FOR i := 1 TO fbSlotList.P_nCount BY 1 DO
	pSlot := fbSlotList.M_GetNext();
	IF pSlot > 0 THEN
		nCurrentPropIndex := nCurrentPropIndex + 1;
		refCmdData.n32Data[nCurrentPropIndex] := pSlot^.P_nNr;
		nCurrentPropIndex := nCurrentPropIndex + 1;
		refCmdData.n32Data[nCurrentPropIndex] := REAL_TO_DINT(pSlot^.P_rRelPosX);
		nCurrentPropIndex := nCurrentPropIndex + 1;
		refCmdData.n32Data[nCurrentPropIndex] := REAL_TO_DINT(pSlot^.P_rRelPosY);
		nCurrentPropIndex := nCurrentPropIndex + 1;
		refCmdData.n32Data[nCurrentPropIndex] := REAL_TO_DINT(pSlot^.P_rRelPosZ);
		nCurrentPropIndex := nCurrentPropIndex + 1;
		refCmdData.n32Data[nCurrentPropIndex] := REAL_TO_DINT(pSlot^.P_rDimWidth);
		nCurrentPropIndex := nCurrentPropIndex + 1;
		refCmdData.n32Data[nCurrentPropIndex] := REAL_TO_DINT(pSlot^.P_rDimDepth);
	END_IF		
END_FOR

nCurrentPropIndex := nCurrentPropIndex + 1;
refCmdData.n32Data[nCurrentPropIndex] := nValveNrSlot1;
nCurrentPropIndex := nCurrentPropIndex + 1;
refCmdData.n32Data[nCurrentPropIndex] := nValveNrSlot2;
nCurrentPropIndex := nCurrentPropIndex + 1;
refCmdData.n32Data[nCurrentPropIndex] := nPumpNrWaste;
nCurrentPropIndex := nCurrentPropIndex + 1;
refCmdData.n32Data[nCurrentPropIndex] := nBottleNrWaste;
END_METHOD

METHOD M_GetProcData : DINT
VAR_INPUT
	eProcDataType : E_ProcDataType;
END_VAR
END_METHOD

METHOD M_GetRectIsInnerSlot : BOOL
VAR_INPUT
	stRectArea : FB_Rectangle;
END_VAR

VAR
	pSlot : POINTER TO FB_DimSlot;
	stPoint: ST_3DPoint;
	fbRect : FB_Rectangle;
	
	
	END_VAR
//Alle Slots durchlaufen
fbSlotList.M_SetCurrentToHead();
REPEAT
	pSlot := fbSlotList.M_GetNext();
	IF pSlot > 0 THEN
		stPoint := pSlot^.P_stAbsPos;
		fbRect.X1 := stPoint.X;
		fbRect.Y1 := stPoint.Y;
		fbRect.X2 := fbRect.X1 + pSlot^.P_rDimWidth;
		fbRect.Y2 := fbRect.Y1 + pSlot^.P_rDimDepth;  
		IF F_RectInnerRect(stRectArea,fbRect) THEN
			M_GetRectIsInnerSlot := TRUE;
			RETURN;
		END_IF
	END_IF
UNTIL pSlot = 0
END_REPEAT
END_METHOD

METHOD M_GetSlot : POINTER TO FB_Slot
VAR_INPUT
	nSlotNr : UINT;
END_VAR
M_GetSlot := fbSlotList.M_GetAtNr(nSlotNr);
END_METHOD

METHOD M_GetSlotFromChild : POINTER TO FB_Slot
VAR_INPUT
	pObject : POINTER TO FB_Object;
END_VAR

VAR
	pSlot : POINTER TO FB_Slot;
END_VAR
//Die SlotList iterieren und vergleichen ob Objekte übereinstimmen
fbSlotList.M_SetCurrentToHead();
REPEAT
	pSlot := fbSlotList.M_GetNext();
	IF pSlot > 0 THEN
		IF pSlot^.P_pChild = pObject THEN
			M_GetSlotFromChild := pSlot;
			EXIT;
		END_IF
	END_IF
UNTIL pSlot = 0
END_REPEAT
END_METHOD

METHOD M_Reset
bError := FALSE;
bBusy := FALSE;
eCurrentState := E_MachineState.MACHINESTATE_Idle;
END_METHOD

METHOD M_SetAllProps : ERRORID
VAR_INPUT
	refCmdData : REFERENCE TO  ST_CmdData;
END_VAR

VAR
	i : UINT;
END_VAR
M_SetAllProps := SUPER^.M_SetAllProps(refCmdData);

IF M_SetAllProps > 0 THEN
	RETURN;
END_IF

//Slots parametrieren
nCurrentPropIndex := nCurrentPropIndex + 1;
nFirstSlotPropIndex := nCurrentPropIndex;
nNumberOfSlots := DINT_TO_UINT(refCmdData.n32Data[nCurrentPropIndex]);

//Falls SlotList noch nicht existiert, dann neue erstellen
IF fbSlotList.P_nCount = 0 THEN
	FOR i:= 1 TO nNumberOfSlots BY 1 DO
		pSlot := __NEW(FB_DimSlot(pOwner := THIS));
		fbSlotList.M_Add(pSlot);
		nCurrentPropIndex := nCurrentPropIndex + 1;
		pSlot^.P_nNr := DINT_TO_USINT(refCmdData.n32Data[nCurrentPropIndex]);
		nCurrentPropIndex := nCurrentPropIndex + 1;
		pSlot^.P_rRelPosX := DINT_TO_REAL(refCmdData.n32Data[nCurrentPropIndex]);
		nCurrentPropIndex := nCurrentPropIndex + 1;
		pSlot^.P_rRelPosY := DINT_TO_REAL(refCmdData.n32Data[nCurrentPropIndex]);
		nCurrentPropIndex := nCurrentPropIndex + 1;
		pSlot^.P_rRelPosZ := DINT_TO_REAL(refCmdData.n32Data[nCurrentPropIndex]);
		nCurrentPropIndex := nCurrentPropIndex + 1;
		pSlot^.P_rDimWidth := DINT_TO_REAL(refCmdData.n32Data[nCurrentPropIndex]);
		nCurrentPropIndex := nCurrentPropIndex + 1;
		pSlot^.P_rDimDepth := DINT_TO_REAL(refCmdData.n32Data[nCurrentPropIndex]);
	END_FOR
ELSE
	IF nNumberOfSlots <> fbSlotList.P_nCount THEN	//Anzahl der Slots dürfen sich nicht ändern
		M_SetAllProps := E_ErrorIdObjMgmt.ERRORID_ChangeNoOfSlotsNotAllowed;
		RETURN;		
	END_IF

	FOR i:= 1 TO nNumberOfSlots BY 1 DO
		nCurrentPropIndex := nCurrentPropIndex + 1;
		pSlot := fbSlotList.M_GetAtNr(DINT_TO_USINT(refCmdData.n32Data[nCurrentPropIndex]));
		IF pSlot > 0 THEN
			nCurrentPropIndex := nCurrentPropIndex + 1;
			pSlot^.P_rRelPosX := DINT_TO_REAL(refCmdData.n32Data[nCurrentPropIndex]);
			nCurrentPropIndex := nCurrentPropIndex + 1;
			pSlot^.P_rRelPosY := DINT_TO_REAL(refCmdData.n32Data[nCurrentPropIndex]);
			nCurrentPropIndex := nCurrentPropIndex + 1;
			pSlot^.P_rRelPosZ := DINT_TO_REAL(refCmdData.n32Data[nCurrentPropIndex]);
			nCurrentPropIndex := nCurrentPropIndex + 1;
			pSlot^.P_rDimWidth := DINT_TO_REAL(refCmdData.n32Data[nCurrentPropIndex]);
			nCurrentPropIndex := nCurrentPropIndex + 1;
			pSlot^.P_rDimDepth := DINT_TO_REAL(refCmdData.n32Data[nCurrentPropIndex]);
		ELSE
			M_SetAllProps := 222;
			RETURN;
		END_IF	
	END_FOR
END_IF
nLastSlotPropIndex := nCurrentPropIndex;
nNoOfProps := nCurrentPropIndex + 1;

nCurrentPropIndex := nCurrentPropIndex + 1;
nSpecPropIndex := nCurrentPropIndex;

nValveNrSlot1 := DINT_TO_USINT(refCmdData.n32Data[nCurrentPropIndex]);
IF NOT (nValveNrSlot1 > 0 AND nValveNrSlot1 <= cNoOfValves) THEN
	M_SetAllProps := E_ErrorIdObjMgmt.ERRORID_InvalidValveNumber;
	RETURN;
END_IF

nCurrentPropIndex := nCurrentPropIndex + 1;
nValveNrSlot2 := DINT_TO_USINT(refCmdData.n32Data[nCurrentPropIndex]);
IF NOT (nValveNrSlot1 > 0 AND nValveNrSlot1 <= cNoOfValves) THEN
	M_SetAllProps := E_ErrorIdObjMgmt.ERRORID_InvalidValveNumber;
	RETURN;
END_IF

nCurrentPropIndex := nCurrentPropIndex + 1;
nPumpNrWaste := DINT_TO_USINT(refCmdData.n32Data[nCurrentPropIndex]);
IF NOT (nPumpNrWaste > 0 AND nPumpNrWaste <= cNoOfPumps) THEN
	M_SetAllProps := E_ErrorIdObjMgmt.ERRORID_InvalidPumpNumber;
	RETURN;
END_IF

nCurrentPropIndex := nCurrentPropIndex + 1;
nBottleNrWaste := DINT_TO_USINT(refCmdData.n32Data[nCurrentPropIndex]);
IF NOT (nBottleNrWaste > 0 AND nBottleNrWaste <= cNoOfWasteBottles) THEN
	M_SetAllProps := E_ErrorIdObjMgmt.ERRORID_InvalidWastebottle;
	RETURN;
END_IF

nNoOfProps := nCurrentPropIndex + 1;
END_METHOD

METHOD M_SetSingleProp : ERRORID
VAR_INPUT
	refCmdData : REFERENCE TO  ST_CmdData;
END_VAR

VAR
	i : UINT;
	nIndex					: UINT;
	nIndexRinseChannels	 	: UINT;
	nIndexWashPoints 	 	: UINT;
	nIndexRestProps 	 	: UINT;
END_VAR
(*nIndexRinseChannels := nSpecPropIndex;
nIndexWashPoints := nIndexRinseChannels + nNoOfRinseChannels * 5 + 1;
nIndexRestProps := nIndexWashPoints + nNoOfWashPoints * 4 + 1;

//Section: RinseChannels
IF refCmdData.aHeader[1] > nIndexRinseChannels AND refCmdData.aHeader[1] < nIndexWashPoints THEN
	FOR i:= 1 TO nNoOfRinseChannels BY 1 DO
		//ersten Index innerhalb der Section ermitteln
		nIndex := nIndexRinseChannels + ((i - 1) * 5) + 1;
		IF refCmdData.aHeader[1] = nIndex THEN	//PumpNr
			IF refCmdData.n32Data[0] >= 0 AND refCmdData.n32Data[0] <= cNoOfPumps THEN
				aStRinseChannels[i].nPumpNr := DINT_TO_USINT(refCmdData.n32Data[0]);
			ELSE
				M_SetSingleProp := E_ErrorIdCmd.ERRORID_InvalidPumpNr;
				RETURN;
			END_IF
			RETURN;
		ELSIF refCmdData.aHeader[1] = nIndex + 1 THEN	//ValveNr
			IF refCmdData.n32Data[0] >= 0 AND refCmdData.n32Data[0] <= cNoOfValves THEN
				aStRinseChannels[i].nValveNr := DINT_TO_USINT(refCmdData.n32Data[0]);
			ELSE
				M_SetSingleProp := E_ErrorIdObjMgmt.ERRORID_InvalidValveNumber;
				RETURN;
			END_IF
		ELSIF refCmdData.aHeader[1] = nIndex + 2 THEN	//StartSpeed in %
			aStRinseChannels[i].nStartSpeed := DINT_TO_USINT(refCmdData.n32Data[0]);	
		ELSIF refCmdData.aHeader[1] = nIndex + 3 THEN	//RatedSpeed in %
			aStRinseChannels[i].nRatedSpeed := DINT_TO_USINT(refCmdData.n32Data[0]);
		ELSIF refCmdData.aHeader[1] = nIndex + 4 THEN	//StartTime in ms
			aStRinseChannels[i].nStartTime := DINT_TO_UINT(refCmdData.n32Data[0]);
		END_IF		
	END_FOR
//Section: Washpoints	
ELSIF refCmdData.aHeader[1] > nIndexWashPoints AND refCmdData.aHeader[1] < nIndexRestProps THEN
	FOR i:= 1 TO nNoOfWashPoints BY 1 DO
		//ersten Index innerhalb der Section ermitteln
		nIndex := nIndexWashPoints + ((i - 1) * 4) + 1;
		IF refCmdData.aHeader[1] = nIndex THEN
			aStWashPoints[i].X := DINT_TO_REAL(refCmdData.n32Data[0]);
		ELSIF refCmdData.aHeader[1] = nIndex + 1 THEN
			aStWashPoints[i].Y := DINT_TO_REAL(refCmdData.n32Data[0]);
		ELSIF refCmdData.aHeader[1] = nIndex + 2 THEN
			aStWashPoints[i].Z := DINT_TO_REAL(refCmdData.n32Data[0]);
		ELSIF refCmdData.aHeader[1] = nIndex + 3 THEN
			M_SetSingleProp := E_ErrorIdCmd.ERRORID_InvalidProperty;
		END_IF			
	END_FOR
//Restliche Props
ELSIF refCmdData.aHeader[1] >= nIndexRestProps AND refCmdData.aHeader[1] < nNoOfProps THEN
	CASE (refCmdData.aHeader[1] - nIndexRestProps) OF
		0: //PumpNrWaste
			IF refCmdData.n32Data[0] > 0 AND refCmdData.n32Data[0] <= cNoOfPumps THEN
				nPumpNrWastePump := DINT_TO_USINT(refCmdData.n32Data[0]);
			ELSE
				M_SetSingleProp := E_ErrorIdCmd.ERRORID_InvalidPumpNr;
			END_IF			
		1: //LiquidBottle
			IF refCmdData.n32Data[0] > 0 AND refCmdData.n32Data[0] <= cNoOfLiquidBottles THEN
				nSysLiquidBottle := DINT_TO_USINT(refCmdData.n32Data[0]);
			ELSE
				M_SetSingleProp := E_ErrorIdObjMgmt.ERRORID_InvalidLiquidbottle;
			END_IF			
		2: //WasteBottle
			IF refCmdData.n32Data[0] > 0 AND refCmdData.n32Data[0] <= cNoOfWasteBottles THEN
				nWasteBottle := DINT_TO_USINT(refCmdData.n32Data[0]);
			ELSE
				M_SetSingleProp := E_ErrorIdObjMgmt.ERRORID_InvalidWastebottle;
			END_IF
		3: //ValveNrDrying (Trockendusche für pH Elektrode)
			IF refCmdData.n32Data[0] >= 0 AND refCmdData.n32Data[0] <= cNoOfValves THEN
				nValveNrAirShower := DINT_TO_USINT(refCmdData.n32Data[0]);
			ELSE
				M_SetSingleProp := E_ErrorIdObjMgmt.ERRORID_InvalidValveNumber;
			END_IF			
	END_CASE	
ELSE
	M_SetSingleProp := SUPER^.M_SetSingleProp(refCmdData);
END_IF*)
END_METHOD

METHOD M_Stop : ERRORID
VAR_INPUT
END_VAR
IF bSuckOff AND nStateA_SuckOff < 70 THEN
	nStateA_SuckOff:= 70;
END_IF
END_METHOD

END_FUNCTION_BLOCK

// ---- Objects/Targets/Active/FB_ActiveTarget.TcPOU
FUNCTION_BLOCK FB_ActiveTarget EXTENDS FB_TargetBase IMPLEMENTS I_Device
VAR_INPUT
END_VAR
VAR_OUTPUT
END_VAR
VAR
	bInitFB			: BOOL := TRUE;
	nNotifyId		: UINT;
	bError			: BOOL;
	nErrorId		: ERRORID;
	bCanceled		: BOOL;
	bStop			: BOOL;
	bBusy			: BOOL;
	eCurrentState	: E_MachineState := E_MachineState.MACHINESTATE_Idle;
	stError			: ST_Error;
	bIsInit			: BOOL;	
	stProcessData	: ST_ObjectProcData;
	eCurrentAction	: E_Action;
	
	//Verkettete Liste für BasicActions
	fbList				: FB_LinkedListCtrl;
	hList				: T_HLINKEDLIST;
	aNodes           	: ARRAY[0..4] OF T_LinkedListEntry;
	getValue			: PVOID;
	getPosPtr       	: POINTER TO T_LinkedListEntry := 0;
	
	
	//Action: "Init"
	bInit				: BOOL;				//Action A_Init() aktiv setzen
	nStateA_Init		: USINT;			//State von A_Init()
	bFlagA_Init			: BOOL := TRUE;		//Hilfsflag A_Init()
	
	//Action: Stop
	nStateA_Stop		: USINT;	//Statemachine von A_Stop()
	bStopAllOnError		: BOOL;
	
	//Action: "Reset"
	nStateA_Reset		: USINT;	//Statemachine von A_Reset();	
END_VAR

METHOD M_CancelAction
VAR_INPUT
	eAction	: E_Action;
END_VAR
END_METHOD

METHOD M_CheckProcDataType : BOOL
VAR_INPUT
	eProcDataType : E_ProcDataType;
END_VAR
END_METHOD

METHOD M_ExeAction : ERRORID
VAR_INPUT
	refActionData	: REFERENCE TO ST_ActionData;
END_VAR
END_METHOD

METHOD M_GetActionBusy : BOOL
VAR_INPUT
	eAction	: E_Action;
END_VAR
END_METHOD

METHOD M_GetAllProps : ERRORID
VAR_INPUT
	refCmdData : REFERENCE TO ST_CmdData;
END_VAR
M_GetAllProps := SUPER^.M_GetAllProps(refCmdData);
refCmdData.aHeader[2] := nNotifyId;
END_METHOD

METHOD M_GetDevice : I_Device
VAR_INPUT
END_VAR
M_GetDevice := THIS^;
END_METHOD

METHOD M_GetProcData : DINT
VAR_INPUT
	eProcDataType : E_ProcDataType;
END_VAR
END_METHOD

METHOD M_Reset
bBusy := TRUE;
eCurrentState := E_MachineState.MACHINESTATE_Reset;
END_METHOD

METHOD M_Stop : ERRORID
//Stop braucht nur ausgeführt werden, wenn irgendwas aktiv ist
IF NOT bStop AND eCurrentState = E_MachineState.MACHINESTATE_Active THEN
	bStop := TRUE;
	fbList.A_AddHeadValue(hList := hList, putValue := E_Action.ACTION_Stop);
END_IF
END_METHOD

PROPERTY P_bBusy : BOOL
GET
P_bBusy := bBusy;
END_GET
END_PROPERTY

PROPERTY P_bCanceled : BOOL
GET
P_bCanceled := bCanceled;
END_GET
END_PROPERTY

PROPERTY P_bError : BOOL
GET
P_bError := bError;
END_GET
END_PROPERTY

PROPERTY P_bIsInit : BOOL
GET
P_bIsInit := bIsInit;
END_GET
END_PROPERTY

PROPERTY P_bStopAllOnError : BOOL
GET
P_bStopAllOnError := bStopAllOnError;
END_GET
END_PROPERTY

PROPERTY P_eCurrentState : E_MachineState
GET
P_eCurrentState := eCurrentState;
END_GET
END_PROPERTY

PROPERTY P_nErrorId : ERRORID
GET
P_nErrorID := nErrorID;
END_GET
END_PROPERTY

PROPERTY P_nNotifyId : UINT
GET
P_nNotifyId := nNotifyId;
END_GET
SET
nNotifyId := P_nNotifyId;
END_SET
END_PROPERTY

PROPERTY P_pObject : POINTER TO FB_Object
GET
P_pObject := THIS;
END_GET
END_PROPERTY

PROPERTY P_stError : ST_Error
GET
P_stError := stError;
END_GET
END_PROPERTY

END_FUNCTION_BLOCK

// ---- Objects/FB_DimSlot.TcPOU
{attribute 'enable_dynamic_creation'}
FUNCTION_BLOCK FB_DimSlot EXTENDS FB_Slot
VAR_INPUT
END_VAR
VAR_OUTPUT
END_VAR
VAR
	stDimension : ST_3DDimension;
END_VAR

PROPERTY P_rDimDepth : REAL
GET
P_rDimDepth := stDimension.Depth;
END_GET
SET
stDimension.Depth := P_rDimDepth;
END_SET
END_PROPERTY

PROPERTY P_rDimHeight : REAL
GET
P_rDimHeight := stDimension.Height;
END_GET
SET
stDimension.Height := P_rDimHeight;
END_SET
END_PROPERTY

PROPERTY P_rDimWidth : REAL
GET
P_rDimWidth := stDimension.Width;
END_GET
SET
stDimension.Width := P_rDimWidth;
END_SET
END_PROPERTY

PROPERTY P_stDimension : ST_3DDimension
GET
P_stDimension := stDimension;
END_GET
SET
stDimension := P_stDimension;
END_SET
END_PROPERTY

END_FUNCTION_BLOCK

// ---- Objects/F_RectInnerRect.TcPOU
FUNCTION F_RectInnerRect : BOOL
VAR_INPUT
	stRect1 : FB_Rectangle;
	stRect2 : FB_Rectangle;
END_VAR
VAR
END_VAR

//Rechteck1 innerhalb Rechteck2?
F_RectInnerRect :=

(stRect1.X1 >= stRect2.X1) AND 
(stRect1.X1 <= stRect2.X2) AND
(stRect1.X2 >= stRect2.X1) AND
(stRect1.X2 <= stRect2.X2) AND

(stRect1.Y1 >= stRect2.Y1) AND 
(stRect1.Y1 <= stRect2.Y2) AND
(stRect1.Y2 >= stRect2.Y1) AND
(stRect1.Y2 <= stRect2.Y2);

END_FUNCTION

// ---- Functions/F_SynchronizeSpeeds.TcPOU
FUNCTION F_SynchronizeSpeeds : ARRAY[0..1] OF REAL;
VAR_INPUT
	rSpeedSum 	: REAL;
	rDistance1 	: REAL;
	rDistance2 	: REAL;
END_VAR
VAR_IN_OUT
	rSpeed1 : REAL;
	rSpeed2 : REAL;
END_VAR
VAR
	rDistSum : REAL;
	rTime : REAL;
END_VAR

//Gesamtweg (Vektor) berechnen
rDistSum := SQRT(rDistance1 * rDistance1 + rDistance2 * rDistance2);
rTime := rDistSum / rSpeedSum;
rSpeed1 := ABS(rDistance1 / rTime);
rSpeed2 := ABS(rDistance2 / rTime);

END_FUNCTION

// ---- Hardware/MultiZ/FB_ZM_Jog.TcPOU
FUNCTION_BLOCK FB_ZM_Jog
VAR_INPUT
	bJogForward		: BOOL;
	bJogBackwards	: BOOL;
	bClock			: BOOL;
	bInching		: BOOL;	//Betriebsart Incremental, es wird um die relative Position bewegt
	pfbZAxisRef		: POINTER TO FB_ZAxisRef;
	rSpeed			: REAL;	//Geschwindigkeit
	rDistance		: REAL;	//relative Distanz, um die in der Betriebsart Incremental verfahren wird
END_VAR

VAR_OUTPUT
	bBusy			: BOOL;
	bError			: BOOL;
	nErrorID		: ERRORID;
END_VAR

VAR
	rTrig1			: R_TRIG;
	fTrig1			: F_TRIG;
	_bClock			: BOOL;
	timeOut			: TON;		//für Betriebsart "Standard" , wenn in dieser Zeitspanne keine neue Flanke kommt, dann Stop
								//verhindert, dass bei einer Unterbrechung der Kommunikation, die Achse unkontrolliert bis an das jeweilige Ende fährt

	bCurrDirForw		: BOOL;		
	bCurrDirBackw		: BOOL;		
	nState				: USINT;
	timeOutErr			: TON;
	rTargetPosition		: REAL;
	nStopReason			: USINT;	//1:regulär 2:timeout clock 3:Richtungswechsel
	nCountStopDirChange : USINT;
END_VAR

IF pfbZAxisRef = 0 THEN
	nErrorId := E_ErrorIdMultiZ.ERRORID_InvalidZChannel;
	bError := TRUE;
	nState := 99;	//go in errorstate		
	RETURN;	
END_IF

//Wird Achse momentan von anderem Movebaustein genutzt?
IF (pfbZAxisRef^.pCurrentFb > 0) AND (pfbZAxisRef^.pCurrentFb <> THIS) THEN //wird von anderem FB genutzt
	RETURN;
END_IF


pfbZAxisRef^.stStatus.bIsMoving := TRUE;

bBusy := TRUE;
fTrig1(CLK:= bJogForward OR bJogBackwards);	//negative Flanke von bJogForward bzw bJogBackwards stoppt
timeOut();	//in der Betriebsart "Standard" muss innerhalb einer gewissen Zeitspanne eine erneute positive Flanke am Eingang kommen, sonst "STOP"

IF pfbZAxisRef^.stInput.nStatus.3 THEN	//Error im Antrieb
	pfbZAxisRef^.stStatus.bError := TRUE;
	bBusy := FALSE;
	pfbZAxisRef^.stOutput.nMode := 0;
	pfbZAxisRef^.stOutput.nCtrl := 0;
	nErrorID := F_MultiZError_TO_ErrorId(pfbZAxisRef^.stInput.nError);
	timeOut(IN:= FALSE);
	bError := TRUE;
	bCurrDirForw := FALSE;
	bCurrDirBackw := FALSE;
	nState := 99;
END_IF

IF timeOutErr.Q THEN
	timeOutErr(IN:= FALSE);
	pfbZAxisRef^.stOutput.nMode := 0;
	pfbZAxisRef^.stOutput.nCtrl := 0;
	CASE nState OF
		2:	//Timeout wait for setpointacknowledge
			nErrorId := E_ErrorIdMultiZ.ERRORID_ToWaitSetPointAck;
		3: //Timeout wait for targetreached
			nErrorId := E_ErrorIdMultiZ.ERRORID_ToWaitTrgtReached;
		6: //Timeout wait for stop
			nErrorId := E_ErrorIdMultiZ.ERRORID_ToWaitStop;
	ELSE
		nErrorId := E_ErrorIdMultiZ.ERRORID_UnknownError;			
	END_CASE
	pfbZAxisRef^.stOutput.nMode := 0;
	pfbZAxisRef^.stOutput.nCtrl := 0;
	bCurrDirForw := FALSE;
	bCurrDirBackw := FALSE;
	bBusy := FALSE;
	bError := TRUE;
	nState := 99;	//go in errorstate
	RETURN;
END_IF

IF NOT bInching AND (bJogForward OR bJogBackwards) THEN	//Betriebsart "Continous"
	IF bClock <> _bClock THEN	//Clock, welcher innerhalb des Timeouts toggeln muss
		rTrig1(CLK:= TRUE);
		_bClock := bClock;
		timeOut(IN:= FALSE);
		timeOut(IN:= TRUE, PT:= T#550MS);		
		//wenn gerade in Move und Richtungsumkehr, dann vorher stoppen
		IF bCurrDirForw AND bJogBackwards THEN	//Richtungsumkehr, stoppen
			nStopReason := 3;
			nState := 5;
		ELSIF bCurrDirBackw AND bJogForward THEN	//Richtungsumkehr, stoppen
			nStopReason := 3;
			nState := 5;
		ELSE
			//Aktuelle Richtung setzen
			IF bJogForward THEN
				bCurrDirForw := TRUE;
				bCurrDirBackw := FALSE;
			ELSIF bJogBackwards THEN
				bCurrDirForw := FALSE;
				bCurrDirBackw := TRUE;
			END_IF			
		END_IF
	ELSE
		IF timeOut.Q THEN	//TiomeOut -> Stoppen
			timeOut(IN:= FALSE);
			nStopReason := 2;
			nstate := 5;	//Stoppen
		END_IF
	END_IF
END_IF

IF fTrig1.Q AND nState > 0  THEN
	timeOut(IN:= FALSE);
	nStopReason := 1;
	nstate := 5;	//Stoppen
END_IF

CASE nState OF
	0:	IF rTrig1.Q THEN
			timeOut(IN:= TRUE, PT:= T#500MS);	//in dieser Zeitzspanne muss eine erneute Flanke kommen, sonst "STOP"
		END_IF
		pfbZAxisRef^.pCurrentFb := THIS; 
		//Geschwindigkeit setzen
		pfbZAxisRef^.stOutput.nVelo := REAL_TO_DINT(rSpeed);
		//Betriebsart Positionsmodus setzen
		pfbZAxisRef^.stOutput.nMode := 1;
		pfbZAxisRef^.stOutput.nCtrl.2 := TRUE; //Relativ

		IF bJogForward THEN //nach oben
			rTargetPosition := pfbZAxisRef^.P_rCurrentPos + rDistance;
			IF rTargetPosition > pfbZAxisRef^.P_rMaxPos THEN
				//Distance anpassen
				rDistance := pfbZAxisRef^.P_rMaxPos - pfbZAxisRef^.P_rCurrentPos;
			END_IF
		ELSE //nach unten
			rTargetPosition := pfbZAxisRef^.P_rCurrentPos - rDistance;
			IF rTargetPosition < pfbZAxisRef^.P_rMinPos THEN
				//Distance anpassen
				rDistance := pfbZAxisRef^.P_rMinPos - pfbZAxisRef^.P_rCurrentPos;
			ELSE
				rDistance := rDistance * -1.0;
			END_IF
		END_IF

		pfbZAxisRef^.P_rRelTargetPos := rDistance;
		
		//Zielposition in Abhängigkeit von Betriebart setzen
		IF NOT bInching THEN	//Betriebsart "Standard" (Continous)
			IF bJogForward THEN //nach oben
				bCurrDirForw := TRUE;
				bCurrDirBackw := FALSE;
			ELSIF bJogBackwards THEN
				bCurrDirForw := FALSE;
				bCurrDirBackw := TRUE;
			END_IF
		END_IF
		
		//Workaround, da FB zweimal im Zyklus aufgerufen wird und Ctrl und Pos im geichen Zyklus auf den CAN-Bus geht
		nState := 10;
		
	1:	//Fahrauftrag starten
		pfbZAxisRef^.stOutput.nCtrl.0 := TRUE;
		nState := 2;
		
	10:	nState := 1;

	2:	//SetpointAcknowledge?
		//Hier könnte es zu einem TimeoutSetpointACK kommen, wenn durch FB_ZMStop Stop das StatusBit nicht kommt
		IF pfbZAxisRef^.stInput.nStatus.1 THEN
			pfbZAxisRef^.stOutput.nCtrl.0 := FALSE;	//Fahrauftrag zuücksetzen
			nState := 3;
			timeOutErr(IN:= FALSE);
		ELSE
			timeOutErr(IN:= TRUE, PT:= T#500MS);
		END_IF
		
	3:	//TargetReached?
		IF pfbZAxisRef^.stInput.nStatus.0 THEN
			rTrig1(CLK:= FALSE);
			_bClock := FALSE;
			nState := 0;	//aktuelle Postion holen
			bBusy := FALSE;
		END_IF
		
	5:	//Stoppen
		pfbZAxisRef^.stOutput.nCtrl.1 := TRUE;	//Stopbit setzen
		pfbZAxisRef^.stOutput.nCtrl.0 := FALSE;	//Fahrauftrag zurücksetzen
		timeOutErr(IN:= FALSE);
 		bCurrDirForw := FALSE;
		bCurrDirBackw := FALSE;		
		nState := 6;
		
	6:	//Stopbit gesetzt?
		IF pfbZAxisRef^.stInput.nStatus.2 THEN
			timeOutErr(IN:= FALSE);
			pfbZAxisRef^.stOutput.nCtrl.1 := FALSE;	//Stopbit zurücksetzen	
			
			pfbZAxisRef^.stOutput.nMode := 0;
				//aus welchem Grund wurde gestoppt?
			IF nStopReason = 1 THEN	//regulär gestoppt
				nState := 0;	//Aktuelle Position holen
				bBusy := FALSE;
			ELSIF nStopReason = 2 THEN //Stop durch timeout
				nState := 0;	//Aktuelle Position holen
				bBusy := FALSE;
			ELSIF nStopReason = 3 THEN //Stop durch Richtungswechsel
				_bClock := NOT _bClock;
				nCountStopDirChange := nCountStopDirChange + 1;
				nState := 0;
			END_IF
		ELSE
			timeOutErr(IN:= TRUE, PT:= T#1000MS);
		END_IF
END_CASE

IF NOT bBusy THEN
	IF pfbZAxisRef^.pCurrentFb = THIS THEN
		pfbZAxisRef^.pCurrentFb := 0;
		pfbZAxisRef^.stStatus.bIsMoving := FALSE;	
	END_IF	
END_IF

METHOD M_Reset
VAR_INPUT
END_VAR
timeOut(IN:= FALSE);
timeOutErr(IN:= FALSE);
rTrig1(CLK:= FALSE);
fTrig1(CLK:= FALSE);
_bClock := FALSE;
bError := FALSE;
nErrorID := 0;
nState := 0;
IF pfbZAxisRef^.pCurrentFb = THIS THEN
	pfbZAxisRef^.pCurrentFb := 0;
	pfbZAxisRef^.stStatus.bIsMoving := FALSE;	
END_IF
END_METHOD

END_FUNCTION_BLOCK

// ---- GCode/FB_Cuboid.TcPOU
FUNCTION_BLOCK FB_Cuboid
VAR_INPUT
END_VAR
VAR_OUTPUT
END_VAR
VAR
	stRefPoint : ST_3DPoint;
	//die  4 Eckpunkte
	aPointsBottom : ARRAY[0..3] OF ST_3DPoint;
	aPointsTop : ARRAY[0..3] OF ST_3DPoint;
	lrAngle: LREAL;	//Verdrehung um Z-Achse
END_VAR

METHOD M_IsPointInnerXY : BOOL
VAR_INPUT
	stTestPoint : ST_3DPoint;
END_VAR
VAR
	A : REAL;	//Fläche
	i : USINT;
	p1 : ST_2DPoint;
	p2 : ST_2DPoint;
	bFlag : BOOL;	
END_VAR
M_IsPointInnerXY := TRUE;
//jeweils mit allen 4 Seiten des Vierecks und dem Testpunkt ein Dreieck bilden und dessen Flächeninhalt berechen (Vektorprodukt)
FOR i := 0 TO 3 BY 1 DO
	p1.X := aPointsBottom[i].X;
	p1.Y := aPointsBottom[i].Y;
	IF i = 3 THEN
		p2.X := aPointsBottom[0].X;
		p2.Y := aPointsBottom[0].Y;
	ELSE
		p2.X := aPointsBottom[i+1].X;
		p2.Y := aPointsBottom[i+1].Y;
	END_IF
	A := 0.5 * (p1.X*p2.Y + p2.X*stTestPoint.Y + stTestPoint.X*p1.Y - p2.X*P1.Y - stTestPoint.X*p2.Y - p1.X*stTestPoint.y);
	IF A < 0.0 THEN
		M_IsPointInnerXY := FALSE;
		RETURN;
	END_IF
END_FOR
END_METHOD

METHOD M_SetDimension
VAR_INPUT
	lrX_Min : LREAL;
	lrX_Max : LREAL;
	lrY_Min : LREAL;
	lrY_Max : LREAL;
	lrZ_Min : LREAL;
	lrZ_Max : LREAL;
END_VAR
VAR
	i : USINT;
END_VAR
//in XY den Bereich etwas vergrößern (Rundungsfehler und Encoderschwankungen)
aPointsBottom[0].X := stRefPoint.X + LREAL_TO_REAL(lrX_Min) - 500.0;
aPointsBottom[0].Y := stRefPoint.Y + LREAL_TO_REAL(lrY_Min) - 500.0;
aPointsBottom[0].Z := stRefPoint.Z + LREAL_TO_REAL(lrZ_Min);

aPointsBottom[1].X := stRefPoint.X + LREAL_TO_REAL(lrX_Max) + 500.0;
aPointsBottom[1].Y := stRefPoint.Y + LREAL_TO_REAL(lrY_Min) - 500.0;
aPointsBottom[1].Z := stRefPoint.Z + LREAL_TO_REAL(lrZ_Min);

aPointsBottom[2].X := stRefPoint.X + LREAL_TO_REAL(lrX_Max) + 500.0;
aPointsBottom[2].Y := stRefPoint.Y + LREAL_TO_REAL(lrY_Max) + 500.0;
aPointsBottom[2].Z := stRefPoint.Z + LREAL_TO_REAL(lrZ_Min);

aPointsBottom[3].X := stRefPoint.X + LREAL_TO_REAL(lrX_Min) - 500.0;
aPointsBottom[3].Y := stRefPoint.Y + LREAL_TO_REAL(lrY_Max) + 500.0;
aPointsBottom[3].Z := stRefPoint.Z + LREAL_TO_REAL(lrZ_Min);

//Alle 4 Punkte drehen
FOR i := 0 TO 3 BY 1 DO
	aPointsBottom[i] := F_RotatePoint(aPointsBottom[i],stRefPoint,lrAngle);
	aPointsTop[i] := aPointsBottom[i];
 	aPointsTop[i].Z := stRefPoint.Z + LREAL_TO_REAL(lrZ_Max);
END_FOR
END_METHOD

PROPERTY P_lrAngle : LREAL
SET
lrAngle := P_lrAngle;
END_SET
END_PROPERTY

PROPERTY P_rXMax : REAL
GET
P_rXMax := MAX(MAX(MAX(aPointsBottom[0].X,aPointsBottom[1].X),aPointsBottom[2].X),aPointsBottom[3].X);
END_GET
END_PROPERTY

PROPERTY P_rXMin : REAL
GET
P_rXMin := MIN(MIN(MIN(aPointsBottom[0].X,aPointsBottom[1].X),aPointsBottom[2].X),aPointsBottom[3].X);
END_GET
END_PROPERTY

PROPERTY P_rYMax : REAL
GET
P_rYMax := MAX(MAX(MAX(aPointsBottom[0].Y,aPointsBottom[1].Y),aPointsBottom[2].Y),aPointsBottom[3].Y);
END_GET
END_PROPERTY

PROPERTY P_rYMin : REAL
GET
P_rYMin := MIN(MIN(MIN(aPointsBottom[0].Y,aPointsBottom[1].Y),aPointsBottom[2].Y),aPointsBottom[3].Y);
END_GET
END_PROPERTY

PROPERTY P_rZMax : REAL
GET
P_rZMax := aPointsTOP[0].Z;
END_GET
END_PROPERTY

PROPERTY P_rZMin : REAL
GET
P_rZMin := aPointsBottom[0].Z;
END_GET
END_PROPERTY

PROPERTY P_stRefPoint : ST_3DPoint
GET
P_stRefPoint := stRefPoint;
END_GET
SET
stRefPoint := P_stRefPoint;
END_SET
END_PROPERTY

END_FUNCTION_BLOCK

// ---- Objects/F_RotatePoint.TcPOU
FUNCTION F_RotatePoint : ST_3DPoint //Rotiert einen Punkt um einen Mittelpunkt in XY-Ebene
VAR_INPUT
	stPoint 	: ST_3DPoint;	//zu rotierender Punkt
	stPointM 	: ST_3DPoint;	//Mittelpunkt
	lrAngle 		: LREAL;	//Drehwinkel
END_VAR
VAR
	lrAngleRad 	: LREAL; //Winkel im Bogenmaß
	stLocVector : ST_2DPoint;
END_VAR

//Ortsvektor von Punkt bilden 
stLocVector.X := stPoint.X - stPointM.X;
stLocVector.Y := stPoint.Y - stPointM.Y;

lrAngleRad := DEG_TO_RAD(lrAngle);
F_RotatePoint.X := LREAL_TO_REAL(stLocVector.X * COS(lrAngleRad) - stLocVector.Y * SIN(lrAngleRad) + stPointM.X); 
F_RotatePoint.Y := LREAL_TO_REAL(stLocVector.X * SIN(lrAngleRad) + stLocVector.Y * COS(lrAngleRad) + stPointM.Y);
F_RotatePoint.Z := stPoint.Z;

END_FUNCTION

// ---- Objects/Pieces/FB_Nozzle.TcPOU
{attribute 'enable_dynamic_creation'}
FUNCTION_BLOCK FB_Nozzle EXTENDS FB_PieceBase
VAR_INPUT
END_VAR
VAR_OUTPUT
END_VAR
VAR
	nCleaningDepth	: DINT;
END_VAR

METHOD FB_init : BOOL
VAR_INPUT
	bInitRetains : BOOL; // if TRUE, the retain variables are initialized (warm start / cold start)
	bInCopyCode : BOOL;  // if TRUE, the instance afterwards gets moved into the copy code (online change)
END_VAR
eObjectType := E_ObjectType.OBJECTTYPE_Nozzle;
eObjectGroup := E_ObjectGroup.OBJECTGROUP_Piece;
END_METHOD

METHOD M_GetAllProps : ERRORID
VAR_INPUT
	refCmdData : REFERENCE TO  ST_CmdData;
END_VAR
SUPER^.M_GetAllProps(refCmdData);
nCurrentPropIndex := nCurrentPropIndex + 1;
refCmdData.n32Data[nCurrentPropIndex] := nCleaningDepth;
END_METHOD

{attribute 'object_name' := 'M_SetAllProps'}
METHOD M_SetAllProps : ERRORID
VAR_INPUT
	refCmdData	: REFERENCE TO ST_CmdData;
END_VAR
M_SetAllProps := SUPER^.M_SetAllProps(refCmdData);

IF M_SetAllProps > 0 THEN
	RETURN;
END_IF
nCurrentPropIndex := nCurrentPropIndex + 1;
nSpecPropIndex := nCurrentPropIndex;

nCleaningDepth := refCmdData.n32Data[nCurrentPropIndex];

nNoOfProps := nCurrentPropIndex + 1;
END_METHOD

METHOD M_SetSingleProp : ERRORID
VAR_INPUT
	refCmdData : REFERENCE TO  ST_CmdData;
END_VAR
IF refCmdData.aHeader[1] = nSpecPropIndex THEN
	nCleaningDepth := refCmdData.n32Data[0];	
ELSE
	M_SetSingleProp := SUPER^.M_SetSingleProp(refCmdData);
END_IF
END_METHOD

PROPERTY P_nCleaningDepth : DINT
GET
P_nCleaningDepth := nCleaningDepth;
END_GET
END_PROPERTY

END_FUNCTION_BLOCK

// ---- Objects/F_LinesIntersect.TcPOU
FUNCTION F_LinesIntersect : BOOL
VAR_INPUT
	stLine1 : St_Line;
	stLine2 : St_Line;
END_VAR
VAR
END_VAR

F_LinesIntersect := 
(stLine1.X1 < stLine2.X1) AND 
(stLine1.X2 > stLine2.X1) AND
(stLine1.Y1 > stLine2.Y1) AND
(stLine1.Y1 < stLine2.Y2)
OR 
(stLine2.X1 < stLine1.X1) AND 
(stLine2.X2 > stLine1.X1) AND
(stLine2.Y1 > stLine1.Y1) AND
(stLine2.Y1 < stLine1.Y2);

END_FUNCTION

// ---- Objects/Targets/Active/FB_HighVoltTray.TcPOU
FUNCTION_BLOCK FB_HighVoltTray EXTENDS FB_ActiveTarget

VAR
	//Hardware-Verküpfung
	pHighVoltSupplyRef	: POINTER TO FB_HighVoltSupply;
	
	//Prozessdaten
	nVoltageActual		: DINT;
	nCurrentActual		: DINT;	//in 10tel µA (10 enstpr. 1.0µA)

	//Variablen allgemeine Statemachine
	
	bCurrentMonitoring		: BOOL;
	bPwrCutOffTriggered		: BOOL;

	//Spec-Properties
	nVoltageChannel			: USINT;
	nCurrentLimit			: UINT; 		//Strombegrenzung der HV-Quelle //in 10tel µA (10 enstpr. 1.0µA)
	
	nPowerCutOffThreshold	: UINT;			//Stromüberwachung (Automatisches Abschalten bei Erreichen) //in 10tel µA (10 enstpr. 1.0µA)
											//wenn "0" , dann wird nicht überwacht
	tPowerCutOffTime		: TIME; 		//wenn Strom für diese Zeit die Abschaltschwelle überschreitet, dann wird abgeschaltet
	
	//****************************************Aktionvariablen****************************************************
	
	//Action: "SetVoltage"
	nVoltageSetpoint	: USINT;
	
	//Action: "SetCurrent"
	nCurrentSetpoint	: USINT;
	
	//Action: "SwitchVoltage"
	bVoltageOn			: BOOL;
	
	timer : TON;	//Stromüberwachung
	
	
END_VAR

IF pHighVoltSupplyRef = 0 THEN
	RETURN;
END_IF

pFbSafety^.M_MesBoxOn();

//durch Notaus oder Unlock werden die Kanäle ausgeschalten und müssen in jedem Fall
//manuell durch SwitchVoltage wieder eingeschalten werden
IF NOT pHighVoltSupplyRef^.bHVPSAvailable THEN
	pHighVoltSupplyRef^.M_SwitchVoltage(1,FALSE);
	pHighVoltSupplyRef^.M_SwitchVoltage(2,FALSE);
END_IF

//Stromüberwachung
nCurrentActual := pHighVoltSupplyRef^.M_GetCurrent();
IF bCurrentMonitoring AND NOT bPwrCutOffTriggered THEN
	IF nCurrentActual >= nPowerCutOffThreshold THEN
		//Strom muss für eine vorgegebene Zeit die Abschaltschwelle erreicht haben.
		timer(IN:= TRUE, PT:= tPowerCutOffTime);
		IF timer.Q THEN
			timer(IN:= FALSE);
			bPwrCutOffTriggered := TRUE; 
			pHighVoltSupplyRef^.M_SwitchVoltage(1,FALSE);
			pHighVoltSupplyRef^.M_SwitchVoltage(2,FALSE);
			stError.POU := E_POU.POU_FB_HighVoltTray;
			stError.ErrorId := E_ErrorIdCmd.ERRORID_OverCurrentHighVoltTray;
			stError.ObjectId := nObjectID;
			fbErrorList.M_Add(stError);			
		END_IF
	ELSE
		timer(IN:= FALSE);
	END_IF
END_IF

//Prozessdaten aktualisieren
stProcessData.nObjId := nObjectID;
stProcessData.n32Data[0] := BOOL_TO_DINT(bIsInit);
stProcessData.n32Data[1] := eCurrentState;
stProcessData.n32Data[2] := stError.ErrorId;

IF nVoltageChannel = 1 THEN
	stProcessData.n32Data[3] := BOOL_TO_DINT(NOT pHighVoltSupplyRef^.bDigiOutVoltage1);
ELSIF nVoltageChannel = 2 THEN
	stProcessData.n32Data[3] := BOOL_TO_DINT(NOT pHighVoltSupplyRef^.bDigiOutVoltage2);
END_IF

nVoltageActual := pHighVoltSupplyRef^.M_GetVoltage();
stProcessData.n32Data[4] := nVoltageActual;
stProcessData.n32Data[5] := nCurrentActual;

aObjProcData[nNotifyId] := stProcessData;

METHOD FB_init : BOOL
VAR_INPUT
	bInitRetains : BOOL; // if TRUE, the retain variables are initialized (warm start / cold start)
	bInCopyCode : BOOL;  // if TRUE, the instance afterwards gets moved into the copy code (online change)
END_VAR
eObjectType := E_ObjectType.OBJECTTYPE_HighVoltTray;
eObjectGroup := E_ObjectGroup.OBJECTGROUP_Target OR E_ObjectGroup.OBJECTGROUP_Device;
END_METHOD

METHOD M_CheckProcDataType : BOOL
VAR_INPUT
	eProcDataType : E_ProcDataType;
END_VAR
IF eProcDataType = E_ProcDataType.PROCDATATYPE_Voltage1 OR eProcDataType = E_ProcDataType.PROCDATATYPE_Current1 THEN
	M_CheckProcDataType := TRUE;
END_IF
END_METHOD

METHOD M_CurrentMonitoring
VAR_INPUT
	bOn : BOOL;
END_VAR
IF bOn THEN
	IF nPowerCutOffThreshold > 0 THEN
		bCurrentMonitoring := TRUE;		
	END_IF
ELSE
	bCurrentMonitoring := FALSE;
 	bPwrCutOffTriggered := FALSE;
END_IF
END_METHOD

METHOD M_ExeAction : ERRORID
VAR_INPUT
	refActionData	: REFERENCE TO ST_ActionData;	
END_VAR
CASE refActionData.eAction OF
	E_Action.ACTION_Init:
		bIsInit := TRUE;
		RETURN;
	E_Action.ACTION_SetVoltage:
		IF 	pHighVoltSupplyRef > 0 THEN
			pHighVoltSupplyRef^.M_SetVoltage(DINT_TO_INT(refActionData.aParams[1]));
			pHighVoltSupplyRef^.M_SetCurrent(nCurrentLimit);
		END_IF
	E_Action.ACTION_SwitchVoltage:
		IF 	pHighVoltSupplyRef > 0 THEN
			IF pHighVoltSupplyRef^.bHVPSAvailable THEN
				pHighVoltSupplyRef^.M_SwitchVoltage(nVoltageChannel,DINT_TO_BOOL(refActionData.aParams[1]));
			ELSE
				M_ExeAction := E_ErrorIdCmd.ERRORID_HighVoltSupplyOff;
			END_IF
		ELSE
			M_ExeAction := E_ErrorIdObjMgmt.ERRORID_InvalidHardwareRef;
		END_IF
	ELSE
		M_ExeAction := E_ErrorIdCmd.ERRORID_InvalidAction;	
END_CASE
END_METHOD

METHOD M_GetActionBusy : BOOL
VAR_INPUT
	eAction : E_Action;
END_VAR
IF eAction = eCurrentAction THEN
	M_GetActionBusy := TRUE;
END_IF
END_METHOD

METHOD M_GetAllProps : ERRORID
VAR_INPUT
	refCmdData : REFERENCE TO  ST_CmdData;
END_VAR
SUPER^.M_GetAllProps(refCmdData);
nCurrentPropIndex := nCurrentPropIndex + 1;
refCmdData.n32Data[nCurrentPropIndex] := nVoltageChannel;
nCurrentPropIndex := nCurrentPropIndex + 1;
refCmdData.n32Data[nCurrentPropIndex] := nCurrentLimit;
nCurrentPropIndex := nCurrentPropIndex + 1;
refCmdData.n32Data[nCurrentPropIndex] := nPowerCutOffThreshold;
nCurrentPropIndex := nCurrentPropIndex + 1;
refCmdData.n32Data[nCurrentPropIndex] := TIME_TO_DINT(tPowerCutOffTime);
END_METHOD

METHOD M_GetProcData : DINT
VAR_INPUT
	eProcDataType : E_ProcDataType;
END_VAR
IF eProcDataType = E_ProcDataType.PROCDATATYPE_Voltage1 THEN
	M_GetProcData := pHighVoltSupplyRef^.M_GetVoltage();
ELSIF eProcDataType = E_ProcDataType.PROCDATATYPE_Current1 THEN
	M_GetProcData := pHighVoltSupplyRef^.M_GetCurrent();
END_IF
END_METHOD

METHOD M_Reset
bBusy := TRUE;
eCurrentState := E_MachineState.MACHINESTATE_Reset;
M_CurrentMonitoring(FALSE);
END_METHOD

METHOD M_SetAllProps : ERRORID
VAR_INPUT
	refCmdData : REFERENCE TO  ST_CmdData;
END_VAR
M_SetAllProps := SUPER^.M_SetAllProps(refCmdData);

IF M_SetAllProps > 0 THEN
	RETURN;
END_IF

{IF defined (variable:fbHighVoltSupplyRef)}
pHighVoltSupplyRef := ADR(fbHighVoltSupplyRef);
{ELSE}
{warning 'implement errorId}
M_SetAllProps := E_ErrorIdObjMgmt.ERRORID_InvalidHardwareRef;
{END_IF}
nCurrentPropIndex := nCurrentPropIndex + 1;
nSpecPropIndex := nCurrentPropIndex;
IF refCmdData.n32Data[nCurrentPropIndex] >= 1 AND refCmdData.n32Data[nCurrentPropIndex] <= 2 THEN
	nVoltageChannel := DINT_TO_USINT(refCmdData.n32Data[nCurrentPropIndex]);
ELSE
	M_SetAllProps := E_ErrorIdObjMgmt.ERRORID_InvalidHardwareRef;
END_IF

nCurrentPropIndex := nCurrentPropIndex + 1;
nCurrentLimit := DINT_TO_UINT(refCmdData.n32Data[nCurrentPropIndex]);
nCurrentPropIndex := nCurrentPropIndex + 1;
nPowerCutOffThreshold := DINT_TO_UINT(refCmdData.n32Data[nCurrentPropIndex]);
nCurrentPropIndex := nCurrentPropIndex + 1;
tPowerCutOffTime := DINT_TO_TIME(refCmdData.n32Data[nCurrentPropIndex]);

nNoOfProps := nCurrentPropIndex + 1;
END_METHOD

METHOD M_SetSingleProp : ERRORID
VAR_INPUT
	refCmdData : REFERENCE TO  ST_CmdData;
END_VAR
IF nSpecPropIndex = refCmdData.aHeader[1] THEN
	IF refCmdData.n32Data[0] >= 1 OR refCmdData.n32Data[0] <= 2 THEN
		IF refCmdData.n32Data[0] <> nVoltageChannel THEN
			IF pHighVoltSupplyRef > 0 THEN
				pHighVoltSupplyRef^.M_SwitchVoltage(1,FALSE);
				pHighVoltSupplyRef^.M_SwitchVoltage(2,FALSE); 
			END_IF
			nVoltageChannel := DINT_TO_USINT(refCmdData.n32Data[0]);
		END_IF
	ELSE
		M_SetSingleProp := E_ErrorIdCmd.ERRORID_InvalidVoltageChannel;	
	END_IF
ELSIF (nSpecPropIndex + 1) = refCmdData.aHeader[1] THEN
	nCurrentLimit := DINT_TO_UINT(refCmdData.n32Data[0]);
	IF pHighVoltSupplyRef > 0 THEN
		pHighVoltSupplyRef^.M_SetCurrent(nCurrentLimit);
	END_IF
ELSIF (nSpecPropIndex + 2) = refCmdData.aHeader[1] THEN
	nPowerCutOffThreshold := DINT_TO_UINT(refCmdData.n32Data[0]);
ELSIF (nSpecPropIndex + 3) = refCmdData.aHeader[1] THEN
	tPowerCutOffTime := DINT_TO_TIME(refCmdData.n32Data[0]);
ELSE
	M_SetSingleProp := SUPER^.M_SetSingleProp(refCmdData);
END_IF
END_METHOD

PROPERTY P_bBusy : BOOL
GET
P_bBusy := bBusy;
END_GET
END_PROPERTY

PROPERTY P_bCanceled : BOOL
GET
P_bCanceled := bCanceled;
END_GET
END_PROPERTY

PROPERTY P_bError : BOOL
GET
IF eCurrentState = E_MachineState.MACHINESTATE_Error THEN
	P_bError := TRUE;
END_IF
END_GET
END_PROPERTY

PROPERTY P_bIsInit : BOOL
GET
P_bIsInit := bIsInit;
END_GET
SET
bIsInit := P_bIsInit;
END_SET
END_PROPERTY

PROPERTY P_bPwrCutOffTriggered : BOOL
GET
P_bPwrCutOffTriggered := bPwrCutOffTriggered;
END_GET
END_PROPERTY

PROPERTY P_bStopAllOnError : BOOL
GET
END_GET
END_PROPERTY

PROPERTY P_nCurrentVoltage : DINT
GET
P_nCurrentVoltage := nVoltageActual;
END_GET
END_PROPERTY

PROPERTY P_stError : ST_Error
GET
END_GET
END_PROPERTY

END_FUNCTION_BLOCK

// ---- Hardware/HighVoltSupply/FB_HighVoltSupply.TcPOU
FUNCTION_BLOCK FB_HighVoltSupply
VAR_INPUT
	nAnalogInVoltage	AT %I* : INT;	//muss mit Analogklemme verknüpft werden
	nAnalogInCurrent	AT %I* : INT;	//muss mit Analogklemme verknüpft werden
	bSafeVoltage		AT %I* : BOOL;	//Spannungsfreiheit
	bHVPSAvailable		AT %I* : BOOL;	//HVPS angesteckt und eingeschalten
END_VAR
VAR_OUTPUT
	nAnalogOutVoltage	AT %Q* : INT;	//muss mit Analogklemme verknüpft werden
	nAnalogOutCurrent	AT %Q* : INT;	//muss mit Analogklemme verknüpft werden
	bDigiOutVoltage1	AT %Q* : BOOL := TRUE;
	bDigiOutVoltage2	AT %Q* : BOOL := TRUE;
END_VAR
VAR
	nCurrentChannel	: USINT;
END_VAR

VAR PERSISTENT
	rMinVoltage		: REAL;
	rMaxVoltage		: REAL;
	rMinVoltageCV	: REAL;
	rMaxVoltageCV	: REAL;
	rMinVoltageMV	: REAL;
	rMaxVoltageMV	: REAL;
	rMinCurrent		: REAL;
	rMaxCurrent		: REAL;
	rMinCurrentCV	: REAL;
	rMaxCurrentCV	: REAL;
	rMinCurrentMV	: REAL;
	rMaxCurrentMV	: REAL;
	bLegacy			: BOOL;
END_VAR

VAR CONSTANT
	cVoltageMax		: REAL := 30000;	//maximal einstellbare Spannung in V
	cCurrentMax		: REAL := 30000;	//maximal einstellbarer Strom in µA (max 30µA bzw max 300µA
END_VAR

IF fbSafety.bEmergencyStop THEN
	bDigiOutVoltage1 := bDigiOutVoltage2 := TRUE;
END_IF

PROPERTY P_nMinVoltageCV : DINT
SET
rMinVoltageCV := DINT_TO_REAL(P_nMinVoltageCV);
fbSettings.M_WritePersData();
END_SET
GET
P_nMinVoltageCV := REAL_TO_DINT(rMinVoltageCV);
END_GET
END_PROPERTY

PROPERTY P_nMaxVoltageMV : DINT
SET
rMaxVoltageMV := DINT_TO_REAL(P_nMaxVoltageMV);
fbSettings.M_WritePersData();
END_SET
GET
P_nMaxVoltageMV := REAL_TO_DINT(rMaxVoltageMV);
END_GET
END_PROPERTY

PROPERTY P_nMinCurrentMV : DINT
GET
P_nMinCurrentMV := REAL_TO_DINT(rMinCurrentMV);
END_GET
SET
rMinCurrentMV := DINT_TO_REAL(P_nMinCurrentMV);
fbSettings.M_WritePersData();
END_SET
END_PROPERTY

METHOD M_SetVoltage : INT
VAR_INPUT
	nValue : INT;
END_VAR

VAR
	rAnaOut			: REAL;
END_VAR
rAnaOut := F_YFuncX(rxMin:= rMinVoltage,
					rxMax:= rMaxVoltage,
					ryMin:= rMinVoltageCV,
					ryMax:= rMaxVoltageCV,
					rx:= nValue) * 32767.0 / 10000.0;

nAnalogOutVoltage := REAL_TO_INT(rAnaOut);
END_METHOD

PROPERTY P_nMaxCurrentMV : DINT
GET
P_nMaxCurrentMV := REAL_TO_DINT(rMaxCurrentMV);
END_GET
SET
rMaxCurrentMV := DINT_TO_REAL(P_nMaxCurrentMV);
fbSettings.M_WritePersData();
END_SET
END_PROPERTY

PROPERTY P_nMaxCurrent : DINT
SET
rMaxCurrent := DINT_TO_REAL(P_nMaxCurrent);
fbSettings.M_WritePersData();
END_SET
GET
P_nMaxCurrent := REAL_TO_DINT(rMaxCurrent);
END_GET
END_PROPERTY

METHOD M_SwitchVoltage
VAR_INPUT
	nChannel : USINT;
	bOn : BOOL;
END_VAR
nCurrentChannel := nChannel;
IF bOn THEN
	pFbSafety^.M_MesBoxOn();
END_IF
IF nChannel = 1 THEN
	bDigiOutVoltage1 := NOT bOn;
	bDigiOutVoltage2 := TRUE;
ELSIF nChannel = 2 THEN
	bDigiOutVoltage1 := TRUE;
	bDigiOutVoltage2 := NOT bOn;
ELSE
	RETURN;
END_IF
END_METHOD

PROPERTY P_nMinCurrentCV : DINT
SET
rMinCurrentCV := DINT_TO_REAL(P_nMinCurrentCV);
fbSettings.M_WritePersData();
END_SET
GET
P_nMinCurrentCV := REAL_TO_DINT(rMinCurrentCV);
END_GET
END_PROPERTY

PROPERTY P_nMaxCurrentCV : DINT
SET
rMaxCurrentCV := DINT_TO_REAL(P_nMaxCurrentCV);
fbSettings.M_WritePersData();
END_SET
GET
P_nMaxCurrentCV := REAL_TO_DINT(rMaxCurrentCV);
END_GET
END_PROPERTY

PROPERTY P_nMinCurrent : DINT
SET
rMinCurrent := DINT_TO_REAL(P_nMinCurrent);
fbSettings.M_WritePersData();
END_SET
GET
P_nMinCurrent := REAL_TO_DINT(rMinCurrent);
END_GET
END_PROPERTY

PROPERTY P_nMinVoltageMV : DINT
GET
P_nMinVoltageMV := REAL_TO_DINT(rMinVoltageMV);
END_GET
SET
rMinVoltageMV := DINT_TO_REAL(P_nMinVoltageMV);
fbSettings.M_WritePersData();
END_SET
END_PROPERTY

METHOD M_GetVoltageOk : BOOL
VAR_INPUT
	nChannel : USINT;
	nSetVoltage	: INT;
	nTolerancePlus	: INT;
	nToleranceMinus	: INT;	
END_VAR

VAR
	nCurrentVoltage : DINT;
END_VAR
nCurrentVoltage := M_GetVoltage();

IF (nCurrentVoltage >= nSetVoltage - nToleranceMinus) AND (nCurrentVoltage <= nSetVoltage + nTolerancePlus)THEN
	M_GetVoltageOk := TRUE;
	RETURN;
END_IF
END_METHOD

METHOD M_GetVoltage : DINT
VAR_INPUT
END_VAR

VAR
	rAnaIn	: REAL;
END_VAR
IF bHVPSAvailable THEN
	//Bei der älteren Bauform wird die Spannung von Kanal2 über den zweiten analogen Eingang gemessen, was bei der neueren Bauform die Strommesung ist
	IF bLegacy AND (nCurrentChannel = 2) THEN
		rAnaIn := nAnalogInCurrent;
	ELSE
		rAnaIn := nAnalogInVoltage;
	END_IF
	
	M_GetVoltage := REAL_TO_DINT(F_YFuncX(rxMin:= rMinVoltageMV,
							rxMax:= rMaxVoltageMV,
							ryMin:= rMinVoltage,
							ryMax:= rMaxVoltage,
							rx:= 10000.0 / 32767.0 * rAnaIn));
END_IF
END_METHOD

PROPERTY P_nMaxVoltageCV : DINT
SET
rMaxVoltageCV := DINT_TO_REAL(P_nMaxVoltageCV);
fbSettings.M_WritePersData();
END_SET
GET
P_nMaxVoltageCV := REAL_TO_DINT(rMaxVoltageCV);
END_GET
END_PROPERTY

METHOD M_GetCurrent : DINT
VAR_INPUT
END_VAR

VAR
	rAnaIn	: REAL;
END_VAR
//Bei älterer Bauform gibt es keine Strommessung
IF bLegacy THEN
	RETURN;
END_IF
IF bHVPSAvailable THEN
	rAnaIn := nAnalogInCurrent;
	M_GetCurrent := REAL_TO_DINT(F_YFuncX(rxMin:= rMinCurrentMV,
										rxMax:= rMaxCurrentMV,
										ryMin:= rMinCurrent,
										ryMax:= rMaxCurrent,
										rx:= 10000.0 / 32767.0 * rAnaIn) * 10.0); //Faktor 10.0 da in 10tel µA mit der
																				  //GUI kommuniziert wird
END_IF
END_METHOD

PROPERTY P_bLegacy : BOOL
SET
bLegacy := P_bLegacy;
fbSettings.M_WritePersData();
END_SET
GET
P_bLegacy := bLegacy;
END_GET
END_PROPERTY

METHOD M_SetCurrent : INT
VAR_INPUT
	nValue : UINT;
END_VAR

VAR
	rAnaOut			: REAL;
	rValue			: REAL;
END_VAR
rValue := DINT_TO_REAL(nValue) / 10.0;
rAnaOut := F_YFuncX(rxMin:= rMinCurrent,
					rxMax:= rMaxCurrent,
					ryMin:= rMinCurrentCV,
					ryMax:= rMaxCurrentCV,
					rx:= rValue) * 32767.0 / 10000.0;

nAnalogOutCurrent := REAL_TO_INT(rAnaOut);
END_METHOD

PROPERTY P_nMinVoltage : DINT
SET
rMinVoltage := DINT_TO_REAL(P_nMinVoltage);
fbSettings.M_WritePersData();
END_SET
GET
P_nMinVoltage := REAL_TO_DINT(rMinVoltage);
END_GET
END_PROPERTY

PROPERTY P_nMaxVoltage : DINT
SET
rMaxVoltage := DINT_TO_REAL(P_nMaxVoltage);
fbSettings.M_WritePersData();
END_SET
GET
P_nMaxVoltage := REAL_TO_DINT(rMaxVoltage);
END_GET
END_PROPERTY

END_FUNCTION_BLOCK

// ---- Hardware/FBox/F_YFuncX.TcPOU
FUNCTION F_YFuncX : REAL
VAR_INPUT
	rxMin: REAL;
	rxMax: REAL;
	ryMin: REAL;
	ryMax: REAL;
	rx: REAL;
END_VAR
VAR
	rGain: REAL;
	rResult: REAL;
END_VAR

IF rxMax = rxMin OR ryMax = ryMin THEN	//Unzulässig
	RETURN;	
END_IF

//Gain positiv oder negativ?
IF (rxMax + rxMin < 0) XOR (ryMax + ryMin < 0) THEN	//Gain negativ
	rGain := (ryMin - ryMax) / (rxMax - rxMin);
	rResult := (rx - rxMax) * rGain + ryMin;
ELSE									//Gain positiv
	rGain := (ryMax - ryMin) / (rxMax - rxMin);
	rResult := (rx - rxMin) * rGain + ryMin;
END_IF

F_YFuncX := LIMIT(ryMin,rResult,ryMax);

END_FUNCTION

// ---- Objects/Tools/FB_CartDispenser.TcPOU
FUNCTION_BLOCK FB_CartDispenser EXTENDS FB_GCodeTool IMPLEMENTS I_Dispenser

VAR_OUTPUT
END_VAR
VAR
	
	//Specproperties
	pPneuChannelPress	: POINTER TO FB_PneuChannelRef;
	pPneuChannelVac		: POINTER TO FB_PneuChannelRef;
	
	nDOutChanValvePress	: USINT;	//Digitaler Ausgangskanal MzHead Druckventil
	
	//****************************************Aktionsvariablen****************************************************

	//Action: "SetPressure"
	bSetPress			: BOOL;
	fbSetPress			: FB_SetPressure;

	//Action: "SetVacuum"
	bSetVacuum			: BOOL;
	fbSetVacuum			: FB_SetPressure;

	//Action: "SwitchPressure"
	bSwitchPress		: BOOL;			
	nStateA_SwitchPress	: USINT;		//State von A_SwitchPress()
	eSwitchPressCtrl	: E_PressCtrl;
	tPressTime			: TIME;			//nach dieser Zeit Ventil automatisch wieder zu
	timerPress			: TON;			//Timer für Öffnungszeit Druckventil
	bPressIsOn			: BOOL;
	
	//Action: "Expose"
	bExpose				: BOOL;
	nStateA_Expose		: USINT;
	pExposure			: POINTER TO FB_Exposure;
	
END_VAR

IF eCurrentState = E_MachineState.MACHINESTATE_Active THEN
	
	IF bSetPress THEN
		fbSetPress(pPneuChannelRef:= pPneuChannelPress);
		IF NOT fbSetPress.bBusy THEN
			IF fbSetPress.bError THEN
				bError := TRUE;
				stError.ErrorId := fbSetPress.nErrorId;
				stError.POU := E_POU.POU_FB_CartDispenser;
				fbErrorList.M_Add(stError);
			END_IF
			bSetPress := FALSE;
			fbSetPress(pPneuChannelRef:= pPneuChannelPress, bExecute:= FALSE);
			M_RemoveListEntry(nSearchValue:= E_Action.ACTION_SetPressure);
		END_IF
	END_IF	

	IF bSetVacuum THEN
		fbSetVacuum(pPneuChannelRef:= pPneuChannelVac);
		IF NOT fbSetVacuum.bBusy THEN
			IF fbSetVacuum.bError THEN
				bError := TRUE;
				stError.ErrorId := fbSetVacuum.nErrorId;
				stError.POU := E_POU.POU_FB_CartDispenser;
				fbErrorList.M_Add(stError);
			END_IF
			bSetVacuum := FALSE;
			fbSetVacuum(pPneuChannelRef:= pPneuChannelVac, bExecute:= FALSE);
			M_RemoveListEntry(nSearchValue:= E_Action.ACTION_SetVacuum);
		END_IF
	END_IF	
	
	IF bSwitchPress THEN	//Kartuschendruck einstellen und Ein-bzw. Aus schalten 
		A_SwitchPress();
		IF nStateA_SwitchPress >= 80 THEN
			IF nStateA_SwitchPress >= 99 THEN
				bError := TRUE;
			END_IF
			bSwitchPress := FALSE;
			nStateA_SwitchPress := 0;
			M_RemoveListEntry(nSearchValue:= E_Action.ACTION_SwitchPressure);
		END_IF
	END_IF
	
	IF bExpose THEN
		A_Expose();
		IF nStateA_Expose >= 80 THEN
			IF nStateA_Expose >= 99 THEN
				bError := TRUE;
			END_IF
			bExpose := FALSE;
			nStateA_Expose := 0;
			M_RemoveListEntry(nSearchValue:= E_Action.ACTION_Expose);
		END_IF
	END_IF
END_IF

SUPER^();	//FB_MzTool aufrufen

IF pPneuChannelPress > 0 THEN
	stProcessData.n32Data[7] := pPneuChannelPress^.P_nCurrentPressure;
END_IF

IF pPneuChannelVac > 0 THEN
	stProcessData.n32Data[8] := pPneuChannelVac^.P_nCurrentPressure;
END_IF

IF pFbMultiZ > 0 THEN
	IF nDOutChanValvePress > 0 AND nDOutChanValvePress < 8 THEN
		bPressIsOn := pFbMultiZ^.aDigiOut[nDOutChanValvePress];
		stProcessData.n32Data[9] := BOOL_TO_DINT(bPressIsOn);
	END_IF
END_IF

aObjProcData[nNotifyId] := stProcessData;

ACTION A_Expose:
IF nStateA_Expose = 70 THEN
	pExposure^.M_CancelAction(ACTION_Expose);
	nStateA_Expose := 71;
END_IF

IF NOT pExposure^.M_GetActionBusy(E_Action.ACTION_Expose) THEN
	nStateA_Expose := 80;
END_IF
END_ACTION

ACTION A_Reset:
//Ist noch eine Aktion aktiv?
IF nStateA_ResetSpec = 0 THEN 
	IF bSetPress THEN
		bSetPress := FALSE;
		fbSetPress(bExecute:= FALSE, pPneuChannelRef:= pPneuChannelPress);
	END_IF

	IF bSetVacuum THEN
		bSetVacuum := FALSE;
		fbSetVacuum(bExecute:= FALSE, pPneuChannelRef:= pPneuChannelVac);
	END_IF
	
	IF bSwitchPress THEN 
		bSwitchPress := FALSE;
		nStateA_SwitchPress := 0;
	END_IF
	nStateA_ResetSpec := 80;		
END_IF

SUPER^.A_Reset();
END_ACTION

ACTION A_Stop:
IF nStateA_Stop = 0 THEN
	
	IF bSetPress THEN
		fbSetPress(bExecute:= FALSE, pPneuChannelRef:= pPneuChannelPress);
	END_IF

	IF bSetVacuum THEN
		fbSetVacuum(bExecute:= FALSE, pPneuChannelRef:= pPneuChannelVac);
	END_IF
	
	IF bSwitchPress AND nStateA_SwitchPress < 70 THEN
		nStateA_SwitchPress := 70;
	END_IF
	
	IF bExpose AND nStateA_Expose < 70 THEN
		nStateA_Expose := 70;
	END_IF
	
	nStateA_Stop := 1;
END_IF

SUPER^.A_Stop();
END_ACTION

ACTION A_SwitchPress:
CASE nStateA_SwitchPress OF
	0:	//Ventil Einschalten
		IF eSwitchPressCtrl = E_PressCtrl.PRESSCTRL_PressOn THEN
			pFbMultiZ^.M_SetDigiOut(nChannel:= nDOutChanValvePress, bValue:= TRUE);
		END_IF
	
		//Timer starten
		IF tPressTime = T#0S THEN
			nStateA_SwitchPress := 80;
			RETURN;	
		END_IF
		
		timerPress(IN:= FALSE);
		timerPress(IN:= TRUE, PT:= tPressTime);
		nStateA_SwitchPress := 1;
		
	1:	//Warten bis Zeitabgelaufen
		timerPress();
		IF timerPress.Q THEN
			timerPress(IN:= FALSE);
			pFbMultiZ^.M_SetDigiOut(nChannel:= nDOutChanValvePress, bValue:= FALSE);
			nStateA_SwitchPress := 80;
		END_IF
		
	70:	//Abbrechen
		timerPress(IN:= FALSE);
		pFbMultiZ^.M_SetDigiOut(nChannel:= nDOutChanValvePress, bValue:= FALSE);
		nStateA_SwitchPress := 80;
END_CASE

//Errorhandling
(*IF nStateA_SwitchPress = 99 THEN
	stError.POU := E_POU.POU_FB_CartridgeDisp;
	stError.Cmd := E_Action.ACTION_SwitchPressure;
	stError.POUAction := E_POUACT.POUACT_A_SwitchPress;
	fbErrorList.M_Add(stError);
END_IF*)
END_ACTION

METHOD FB_init : BOOL
VAR_INPUT
	bInitRetains : BOOL; // if TRUE, the retain variables are initialized (warm start / cold start)
	bInCopyCode : BOOL;  // if TRUE, the instance afterwards gets moved into the copy code (online change)
END_VAR
eObjectType := E_ObjectType.OBJECTTYPE_CartDispenser;
eObjectGroup := E_ObjectGroup.OBJECTGROUP_MzTool OR E_ObjectGroup.OBJECTGROUP_Device;
END_METHOD

METHOD M_AddChild : ERRORID
VAR_INPUT
	pObject : POINTER TO FB_Object;
	nSlotNr	: UINT;
	nIndex : INT;
END_VAR
IF pObject > 0 THEN
	IF pObject^.P_eObjectType = E_ObjectType.OBJECTTYPE_Nozzle THEN
		M_AddChild := SUPER^.M_AddChild(pObject,nSlotNr,nIndex);
	ELSE
		M_AddChild := E_ErrorIdObjMgmt.ERRORID_InvalidParentObject;
	END_IF
ELSE
	M_AddChild := E_ErrorIdObjMgmt.ERRORID_InvalidParentObject;
END_IF
END_METHOD

METHOD M_CancelAction
VAR_INPUT
	eAction : E_Action;
END_VAR
CASE eAction OF
	E_Action.ACTION_SetPressure:
		IF bSetPress THEN
			fbSetPress(bExecute:= FALSE, pPneuChannelRef:= pPneuChannelPress);
		END_IF
	
	E_Action.ACTION_SetVacuum:
		IF bSetVacuum THEN
			fbSetVacuum(bExecute:= FALSE, pPneuChannelRef:= pPneuChannelVac);
		END_IF
	
	E_Action.ACTION_SwitchPressure:
		IF bSwitchPress AND nStateA_SwitchPress < 70 THEN
			nStateA_SwitchPress := 70;
		END_IF

	E_Action.ACTION_Expose:
		IF bExpose AND nStateA_Expose < 70 THEN
			nStateA_Expose := 70;
		END_IF
ELSE
	SUPER^.M_CancelAction(eAction);
END_CASE
END_METHOD

METHOD M_CheckAction : ERRORID
VAR_INPUT
	refActionData : REFERENCE TO ST_ActionData;
	pCorrelObject	: POINTER TO FB_Object;
END_VAR
CASE refActionData.eAction OF
	E_Action.ACTION_CleanTip,
	E_Action.ACTION_MeasureTool,
	E_Action.ACTION_SwitchPressure, //BasicAction für ActionOnArray
	E_Action.ACTION_TeachTarget:
		RETURN;
ELSE
	M_CheckAction := SUPER^.M_CheckAction(refActionData, pCorrelObject);
END_CASE
END_METHOD

METHOD M_CheckProcDataType : BOOL
VAR_INPUT
	eProcDataType : E_ProcDataType;
END_VAR
IF eProcDataType = E_ProcDataType.PROCDATATYPE_Temp1 OR eProcDataType = E_ProcDataType.PROCDATATYPE_Press1 THEN
	M_CheckProcDataType := TRUE;
END_IF
END_METHOD

METHOD M_CheckProps : ERRORID
VAR_INPUT
END_VAR

VAR
	iterator : FB_ObjCollectIterator;
	pHybridDispenser : POINTER TO FB_HybridDispenser;
END_VAR
M_CheckProps := SUPER^.M_CheckProps();
//Checken, ob an Holder ein Exposure hängt
pExposure := 0;
pObjCollectNode^.P_pOwnerColl^.M_GetIterator(iterator);
WHILE iterator.pNode > 0 DO
	IF iterator.pNode^.P_pObject^.P_eObjectType = E_ObjectType.OBJECTTYPE_Exposure THEN
		pExposure := iterator.pNode^.P_pObject;
		EXIT;
	END_IF
	iterator.M_Increment();
END_WHILE

//Nozzle muss zwingend dran wenn:
//Parent ist ein CartridgeHolder
//Parent ist ein HybridDispenser und hängt am MasterSlot
IF pPiece = 0 THEN
	IF pParentMzTool^.P_eObjectType = E_ObjectType.OBJECTTYPE_CartHolder THEN
		M_CheckProps := E_ErrorIdObjMgmt.ERRORID_NoNozzleOnTool;
	ELSIF pParentMzTool^.P_eObjectType = E_ObjectType.OBJECTTYPE_HybridDispenser THEN
		pHybridDispenser := pParentMzTool;
		IF pHybridDispenser^.M_ToolIsOnMasterSlot(THIS) THEN
			M_CheckProps := E_ErrorIdObjMgmt.ERRORID_NoNozzleOnTool;
		END_IF
	END_IF	
END_IF
END_METHOD

METHOD M_ClearAllProps
VAR_INPUT
	bIgnoreParent : BOOL; //Es wird das gesamte OD gelöscht. -> Zeiger auf Parent nicht mehr gültig!
END_VAR
pExposure := 0;
pPneuChannelPress := 0;
pPneuChannelVac := 0;
SUPER^.M_ClearAllProps(bIgnoreParent);
END_METHOD

METHOD M_DispenserPrepare : ERRORID
VAR_INPUT
END_VAR
END_METHOD

METHOD M_DispenserStart : ERRORID
VAR_INPUT
END_VAR
IF NOT (eCurrentState = E_MachineState.MACHINESTATE_Idle OR
	eCurrentState = E_MachineState.MACHINESTATE_Active OR
	eCurrentState = E_MachineState.MACHINESTATE_Ready) THEN
	M_DispenserStart := E_ErrorIdCmd.ERRORID_InvalidState;
	RETURN;
END_IF

IF bSwitchPress THEN //ist eventuell durch direkte Action "SwitchPress" mit Time aktiv
	tPressTime := T#0S;
	nStateA_SwitchPress := 0;
ELSE
	pFbMultiZ^.M_SetDigiOut(nChannel:= nDOutChanValvePress, bValue:= TRUE);
END_IF
END_METHOD

METHOD M_DispenserStop : ERRORID
VAR_INPUT
END_VAR
IF bSwitchPress THEN
	nStateA_SwitchPress := 80;
ELSE
	pFbMultiZ^.M_SetDigiOut(nChannel:= nDOutChanValvePress, bValue:= FALSE);
END_IF
END_METHOD

METHOD M_ExeAction : ERRORID
VAR_INPUT
	refActionData : REFERENCE TO ST_ActionData;	
END_VAR
IF NOT (eCurrentState = E_MachineState.MACHINESTATE_Idle OR
	eCurrentState = E_MachineState.MACHINESTATE_Active OR
	eCurrentState = E_MachineState.MACHINESTATE_Ready) THEN
	M_ExeAction := E_ErrorIdCmd.ERRORID_InvalidState;
	RETURN;
END_IF

CASE refActionData.eAction OF
		
	E_Action.ACTION_SetPressure:
		fbSetPress(bExecute:= FALSE, pPneuChannelRef:= pPneuChannelPress); //eventueller Fehler wird auch zurückgesetzt
		fbSetPress.bAwait := DINT_TO_BOOL(refActionData.aParams[1]);
		fbSetPress.nValue := DINT_TO_INT(refActionData.aParams[2]);
		fbSetPress.nTolerancePlus := DINT_TO_INT(refActionData.aParams[3]);
		fbSetPress.nToleranceMinus := DINT_TO_INT(refActionData.aParams[4]);
		fbSetPress.tTimeout := DINT_TO_TIME(refActionData.aParams[5]);
		
		fbSetPress(bExecute:= TRUE,	pPneuChannelRef:= pPneuChannelPress,nErrorId=> M_ExeAction);
		IF fbSetPress.bError THEN
			RETURN;
		END_IF
		
		IF NOT bSetPress AND fbSetPress.bBusy THEN
			bSetPress := TRUE;
			fbList.A_AddHeadValue(hList := hList, putValue := E_Action.ACTION_SetPressure);
		ELSE
			RETURN;	
		END_IF

	E_Action.ACTION_SetVacuum:
		fbSetVacuum(bExecute:= FALSE, pPneuChannelRef:= pPneuChannelVac); //eventueller Fehler wird auch zurückgesetzt
		fbSetVacuum.bAwait := DINT_TO_BOOL(refActionData.aParams[1]);
		fbSetVacuum.nValue := DINT_TO_INT(refActionData.aParams[2]);
		fbSetVacuum.nTolerancePlus := DINT_TO_INT(refActionData.aParams[3]);
		fbSetVacuum.nToleranceMinus := DINT_TO_INT(refActionData.aParams[4]);
		fbSetVacuum.tTimeout := DINT_TO_TIME(refActionData.aParams[5]);
		
		fbSetVacuum(bExecute:= TRUE, pPneuChannelRef:= pPneuChannelVac,nErrorId=> M_ExeAction);
		IF fbSetVacuum.bError THEN
			RETURN;
		END_IF
		
		IF NOT bSetVacuum AND fbSetVacuum.bBusy THEN
			bSetVacuum := TRUE;
			fbList.A_AddHeadValue(hList := hList, putValue := E_Action.ACTION_SetVacuum);
		ELSE
			RETURN;	
		END_IF
		
	E_Action.ACTION_SwitchPressure:
			eSwitchPressCtrl := DINT_TO_USINT(refActionData.aParams[1]);
			IF (eSwitchPressCtrl = E_PressCtrl.PRESSCTRL_PressOn) OR (eSwitchPressCtrl = E_PressCtrl.PRESSCTRL_Off) THEN
				tPressTime := DINT_TO_TIME(refActionData.aParams[2]);
				//Wenn Aktion aktiv kann es sein das die Zeit noch läuft oder der Druck an ist
				IF bSwitchPress THEN	//Aktion ist aktiv
					IF eSwitchPressCtrl = E_PressCtrl.PRESSCTRL_PressOn THEN
						//Statemachine zurücksetzen
						nStateA_SwitchPress := 0;		
					ELSE
						pFbMultiZ^.M_SetDigiOut(nChannel:= nDOutChanValvePress, bValue:= FALSE);
						nStateA_SwitchPress := 80;
					END_IF
				ELSE	//Aktion ist nicht aktiv
					IF eSwitchPressCtrl = E_PressCtrl.PRESSCTRL_PressOn THEN
						bSwitchPress := TRUE;
						fbList.A_AddHeadValue(hList := hList, putValue := E_Action.ACTION_SwitchPressure);
					ELSE
						pFbMultiZ^.M_SetDigiOut(nChannel:= nDOutChanValvePress, bValue:= FALSE);
						RETURN;
					END_IF
				END_IF
			ELSE
				M_ExeAction := E_ErrorIdCmd.ERRORID_InvalidCtrl;
				RETURN;
			END_IF
	
	E_Action.ACTION_Expose:
		//Die Action kann nur über einen Exposer, der als Child an diesem Tool hängt ausgeführt werden
		IF pExposure > 0 THEN
			M_ExeAction := pExposure^.M_ExeAction(refActionData);
			IF M_ExeAction > 0 THEN
				RETURN;
			ELSE
				IF NOT bExpose THEN
					fbList.A_AddHeadValue(hList := hList, putValue := E_Action.ACTION_Expose);	
				END_IF
				bExpose := TRUE;
			END_IF
		ELSE
			M_ExeAction := E_ErrorIdCmd.ERRORID_NoExposureConfigured;
			RETURN;
		END_IF
		
	E_Action.ACTION_BasicDispense:
		IF refActionData.aParams[1] = 0 THEN
			M_ExeAction := M_DispenserStop();
		ELSE
			M_ExeAction := M_DispenserStart();	
		END_IF
		IF M_ExeAction > 0 THEN
			RETURN;
		END_IF
	ELSE
		M_ExeAction := SUPER^.M_ExeAction(refActionData);
		RETURN;
END_CASE

bBusy := TRUE;
eCurrentState := E_MachineState.MACHINESTATE_Active;
END_METHOD

METHOD M_GetAllProps : ERRORID
VAR_INPUT
	refCmdData : REFERENCE TO  ST_CmdData;
END_VAR
//Basisproperties lesen
SUPER^.M_GetAllProps(refCmdData);
//Specialproperties lesen
nCurrentPropIndex := nCurrentPropIndex + 1; 
IF pPneuChannelPress > 0 THEN
	refCmdData.n32Data[nCurrentPropIndex] := pPneuChannelPress^.nChannel;
ELSE
	refCmdData.n32Data[nCurrentPropIndex] := 0;
END_IF

nCurrentPropIndex := nCurrentPropIndex + 1;
IF pPneuChannelVac > 0 THEN
	refCmdData.n32Data[nCurrentPropIndex] := pPneuChannelVac^.nChannel;
ELSE
	refCmdData.n32Data[nCurrentPropIndex] := 0;
END_IF

nCurrentPropIndex := nCurrentPropIndex + 1; 
refCmdData.n32Data[nCurrentPropIndex] := nDOutChanValvePress; //Digitaler Ausgangskanal MzHead Druckventil
nCurrentPropIndex := nCurrentPropIndex + 1; 
refCmdData.n32Data[nCurrentPropIndex] := BOOL_TO_DINT(bIsMESTool);
END_METHOD

METHOD M_GetProcData : DINT
VAR_INPUT
	eProcDataType : E_ProcDataType;
END_VAR
IF eProcDataType = E_ProcDataType.PROCDATATYPE_Press1 THEN
	M_GetProcData := stProcessData.n32Data[7];
END_IF
END_METHOD

METHOD M_SetAllProps : ERRORID
VAR_INPUT
	refCmdData : REFERENCE TO  ST_CmdData;
END_VAR

VAR
	nPneuChannel : USINT;
END_VAR
M_SetAllProps := SUPER^.M_SetAllProps(refCmdData);

IF M_SetAllProps > 0 THEN
	RETURN;
END_IF

//PneuChannel Druck
nCurrentPropIndex := nCurrentPropIndex + 1;
nSpecPropIndex := nCurrentPropIndex;
nPneuChannel := DINT_TO_USINT(refCmdData.n32Data[nCurrentPropIndex]);	//PneuChannel Druck
IF NOT (nPneuChannel > 0 AND nPneuChannel <= cNoOfPneuChannels) THEN
	M_SetAllProps := E_ErrorIdObjMgmt.ERRORID_InvalidPneuChannel;
	RETURN;	
END_IF
pPneuChannelPress := ADR(aFbPneuChannel[nPneuChannel]);

//PneuChannel Vakuum
//Für Vakuum kann der PneuChannel auch auf "0" festgelegt werden. (kein Haltevakkum)
nCurrentPropIndex := nCurrentPropIndex + 1;
nPneuChannel := DINT_TO_USINT(refCmdData.n32Data[nCurrentPropIndex]);		
IF nPneuChannel > 0 AND nPneuChannel <= cNoOfPneuChannels THEN
	pPneuChannelVac := ADR(aFbPneuChannel[nPneuChannel]);
ELSIF nPneuChannel = 0 THEN
	pPneuChannelVac := 0;
ELSE
	M_SetAllProps := E_ErrorIdObjMgmt.ERRORID_InvalidPneuChannel;
	RETURN;	
END_IF

//Digitale Ausgänge auf MzHead müssen zwischen 1 und 7 liegen
nCurrentPropIndex := nCurrentPropIndex + 1;
nDOutChanValvePress := DINT_TO_USINT(refCmdData.n32Data[nCurrentPropIndex]);	//Digitaler Ausgangskanal MzHead Druckventil
IF NOT(nDOutChanValvePress > 0 AND nDOutChanValvePress <= 7) THEN
	M_SetAllProps := E_ErrorIdObjMgmt.ERRORID_InvalidMzDOutChannel;
	RETURN;
END_IF

nCurrentPropIndex := nCurrentPropIndex + 1;
bIsMESTool := DINT_TO_BOOL(refCmdData.n32Data[nCurrentPropIndex]);
nNoOfProps := nCurrentPropIndex + 1;
END_METHOD

METHOD M_SetPrintParams : ST_MethResult
VAR_INPUT
	eType 		: E_PrintParamType;
	nNumerator	: USINT;
	nValue		: DINT;
END_VAR

VAR
	stActionData : ST_ActionData;
END_VAR

VAR_STAT
	bExecuted : BOOL;
END_VAR
IF eType = E_PrintParamType.Pressure THEN
	IF nNumerator <> 1 THEN
		M_SetPrintParams.bError := TRUE;
		M_SetPrintParams.nErrorId := E_ErrorIdCmd.ERRORID_InvalidPrintParamNumerator;
		RETURN;
	END_IF
	
	IF nValue > 1 AND NOT pPneuChannelPress^.P_bSupplyOk THEN 
		M_SetPrintParams.bError := TRUE;
		M_SetPrintParams.nErrorId := E_ErrorIdCmd.ERRORID_PressureSupply;
		RETURN;
	END_IF

	stActionData.eAction := E_Action.ACTION_SetPressure;
	stActionData.aParams[2] := nValue; //Soll
	
	//Überwachung nur, wenn Druck noch nicht an
	//Damit wird verhindert, dass es beim Gradientendruck zu Zeitverzögerungen kommt 
	IF NOT bPressIsOn THEN
		stActionData.aParams[1] := 1; //Fertigmeldung, wenn Druck erreicht
		stActionData.aParams[3] := 20; //Toleranz +
		stActionData.aParams[4] := 20; //Toleranz -
		stActionData.aParams[5] := 20000; //Timeout
	END_IF
	
	IF NOT bExecuted THEN
		M_SetPrintParams.nErrorId := M_ExeAction(stActionData);
		bExecuted := TRUE;
	END_IF
	
	IF M_SetPrintParams.nErrorId > 0 THEN
		M_SetPrintParams.bError := TRUE;
	ELSIF M_GetActionBusy(E_Action.ACTION_SetPressure) THEN //ist ActionStatemachine zur Überwachung gegangen
		M_SetPrintParams.bBusy := TRUE;
		RETURN;
	END_IF
ELSE
	M_SetPrintParams.bError := TRUE;
	M_SetPrintParams.nErrorId := E_ErrorIdCmd.ERRORID_InvalidPrintParamType;
END_IF

bExecuted := FALSE;
END_METHOD

METHOD M_SetSingleProp : ERRORID
VAR_INPUT
	refCmdData : REFERENCE TO  ST_CmdData;
END_VAR

VAR
	nPneuChannel : USINT;
END_VAR
IF nSpecPropIndex = refCmdData.aHeader[1] THEN	//PneuChannelPressure
	nPneuChannel := DINT_TO_USINT(refCmdData.n32Data[0]);
	IF NOT (nPneuChannel > 0 AND nPneuChannel <= cNoOfPneuChannels) THEN
		M_SetSingleProp := E_ErrorIdObjMgmt.ERRORID_InvalidPneuChannel;
		RETURN;	
	END_IF
	pPneuChannelPress := ADR(aFbPneuChannel[nPneuChannel]);
ELSIF nSpecPropIndex + 1 = refCmdData.aHeader[1] THEN	//PneuChannel Vacuum
	nPneuChannel := DINT_TO_USINT(refCmdData.n32Data[0]);
	IF NOT (nPneuChannel >= 0 AND nPneuChannel <= cNoOfPneuChannels) THEN
		M_SetSingleProp := E_ErrorIdObjMgmt.ERRORID_InvalidPneuChannel;
		RETURN;	
	END_IF
	pPneuChannelVac := ADR(aFbPneuChannel[nPneuChannel]);
ELSIF nSpecPropIndex + 2 = refCmdData.aHeader[1] THEN	//Digitaler Ausgangskanal MzHead Druckventil
	IF refCmdData.n32Data[0] >= 0 AND refCmdData.n32Data[0] <= cNoOfValves THEN
		nDOutChanValvePress := DINT_TO_USINT(refCmdData.n32Data[0]);
	ELSE
		M_SetSingleProp := E_ErrorIdObjMgmt.ERRORID_InvalidValveNumber;
	END_IF	
ELSE
	M_SetSingleProp := SUPER^.M_SetSingleProp(refCmdData);
END_IF
END_METHOD

METHOD M_SwitchPressure : ERRORID
VAR_INPUT
	eSwitchPressCtrl : E_PressCtrl;
	tPressTime : TIME;
END_VAR
//Diese Methode funktioniert ähnlich der Methode M_ExeAction, nur dass sie auf SwitchPressure spezialisiert ist
IF NOT (eCurrentState = E_MachineState.MACHINESTATE_Idle OR
	eCurrentState = E_MachineState.MACHINESTATE_Active OR
	eCurrentState = E_MachineState.MACHINESTATE_Ready) THEN
	M_SwitchPressure := E_ErrorIdCmd.ERRORID_InvalidState;
	RETURN;
END_IF

IF (eSwitchPressCtrl = E_PressCtrl.PRESSCTRL_PressOn) OR (eSwitchPressCtrl = E_PressCtrl.PRESSCTRL_Off) THEN
	THIS^.eSwitchPressCtrl := eSwitchPressCtrl;
	THIS^.tPressTime := tPressTime;
	//Wenn Aktion aktiv kann es sein das die Zeit noch läuft oder der Druck an ist
	IF bSwitchPress THEN	//Aktion ist aktiv
		IF eSwitchPressCtrl = E_PressCtrl.PRESSCTRL_PressOn THEN
			//Statemachine zurücksetzen
			nStateA_SwitchPress := 0;		
		ELSE
			pFbMultiZ^.M_SetDigiOut(nChannel:= nDOutChanValvePress, bValue:= FALSE);
			nStateA_SwitchPress := 80;
		END_IF
	ELSE	//Aktion ist nicht aktiv
		IF eSwitchPressCtrl = E_PressCtrl.PRESSCTRL_PressOn THEN
			bSwitchPress := TRUE;
			fbList.A_AddHeadValue(hList := hList, putValue := E_Action.ACTION_SwitchPressure);
		ELSE
			pFbMultiZ^.M_SetDigiOut(nChannel:= nDOutChanValvePress, bValue:= FALSE);
		END_IF
	END_IF
ELSE
	M_SwitchPressure := E_ErrorIdCmd.ERRORID_InvalidCtrl;
	RETURN;
END_IF

bBusy := TRUE;
eCurrentState := E_MachineState.MACHINESTATE_Active;
END_METHOD

PROPERTY P_bPressIsOn : BOOL
GET
P_bPressIsOn := bPressIsOn;
END_GET
END_PROPERTY

PROPERTY P_eDispenserState : E_DispenserState
GET
IF bPressIsOn THEN
	P_eDispenserState := E_DispenserState.Dispensing;	
END_IF
END_GET
END_PROPERTY

PROPERTY P_stCurrentXYArea : FB_RectAngle
GET
VAR
	stPoint : ST_3DPoint;
	stDim	: ST_3DDimension;
END_VAR
stPoint := P_stCurrentPosPhys;
IF pPiece > 0 THEN
	stDim := pPiece^.P_stDimension;
	P_stCurrentXYArea.X1 := stPoint.X - stDim.Width / 2.0;
	P_stCurrentXYArea.X2 := stPoint.X + stDim.Width / 2.0;
	P_stCurrentXYArea.Y1 := stPoint.Y - stDim.Width / 2.0;
	P_stCurrentXYArea.Y2 := stPoint.Y + stDim.Width / 2.0;
ELSE
	P_stCurrentXYArea.X1 := stPoint.X - 1000.0;
	P_stCurrentXYArea.X2 := stPoint.X + 1000.0;
	P_stCurrentXYArea.Y1 := stPoint.Y - 1000.0;
	P_stCurrentXYArea.Y2 := stPoint.Y + 1000.0;	
END_IF
END_GET
END_PROPERTY

END_FUNCTION_BLOCK

// ---- Objects/Tools/FB_GCodeTool.TcPOU
FUNCTION_BLOCK FB_GCodeTool EXTENDS FB_MzTool
VAR_INPUT
END_VAR
VAR_OUTPUT
END_VAR
VAR
	nGCodeToolNr : USINT;
END_VAR

SUPER^();	//FB_MzTool aufrufen

METHOD M_CheckGCodeStart : ERRORID
VAR_INPUT
END_VAR
//Wird derzeit von den Tool überschrieben, die Extruder sind und gelockt werden müssen.
END_METHOD

METHOD M_GetAllProps : ERRORID
VAR_INPUT
	refCmdData : REFERENCE TO  ST_CmdData;
END_VAR
SUPER^.M_GetAllProps(refCmdData);
nCurrentPropIndex := nCurrentPropIndex + 1;
refCmdData.n32Data[nCurrentPropIndex] := nGCodeToolNr;
END_METHOD

METHOD M_SetAllProps : ERRORID
VAR_INPUT
	refCmdData : REFERENCE TO  ST_CmdData;
END_VAR
M_SetAllProps := SUPER^.M_SetAllProps(refCmdData);

IF M_SetAllProps > 0 THEN
	RETURN;
END_IF

nCurrentPropIndex := nCurrentPropIndex + 1;
nSpecPropIndex := nCurrentPropIndex;
nGCodeToolNr := DINT_TO_USINT(refCmdData.n32Data[nCurrentPropIndex]);
nNoOfProps := nCurrentPropIndex + 1;

eObjectGroup := eObjectGroup OR E_ObjectGroup.OBJECTGROUP_GCodeTool;
END_METHOD

METHOD M_SetPrintParams : ST_MethResult
VAR_INPUT
	eType 		: E_PrintParamType;
	nNumerator	: USINT;
	nValue		: DINT;
END_VAR
END_METHOD

METHOD M_StartUniDispense : ERRORID
VAR_INPUT
	nParam1 : DINT;
	nParam2 : DINT;
END_VAR

VAR_OUTPUT
	bIsContinous : BOOL;
END_VAR
M_StartUniDispense := E_ErrorIdGCode.ERRORID_ToolIsNoUniDispenser;
END_METHOD

METHOD M_StopUniDispense : ERRORID
VAR_INPUT
END_VAR
END_METHOD

PROPERTY P_nGCodeToolNr : USINT
GET
P_nGCodeToolNr := nGCodeToolNr;
END_GET
END_PROPERTY

END_FUNCTION_BLOCK

// ---- Hardware/FBox/PneuChannels/FB_PneuChannelRef.TcPOU
FUNCTION_BLOCK FB_PneuChannelRef
VAR_INPUT
	
END_VAR
VAR_OUTPUT
	nSetPress		: INT;		//Solldruck
	nCurrentPress	: INT;		//aktueller Ausgangsdruck in kPa
	nChannel		: USINT;	//Channel-Nr.
END_VAR
VAR
	bSupplyOk		AT %I* : BOOL;	//Druckschalter Versorgung
	nAnalogInput	AT %I* : INT;	//muss mit Analogklemme verknüpft werden
	nAnalogOutput	AT %Q* : INT;	//muss mit Analogklemme verknüpft werden
	bSupplyActor	AT %Q* : BOOL;	//Aktor z.B. Ventil oder Druck-bzw. Vakuumpumpe o.ä.
	nTemp			: DINT;
	bPressOk		: BOOL;	//Druck ist im Toleranzbereich
END_VAR

VAR PERSISTENT
	rMinPress		: REAL;	//minimal einstellbarer Druck/Vacuum des ITV in kPa
	rMaxPress		: REAL;	//maximal einstellbarer Druck/Vacuum des ITV in kPa
	rMinPressCV		: REAL;	//Steuerspannung für "rMinPress" in V
	rMaxPressCV		: REAL;	//Steuerspannung für "rMaxPress" in V
	rMinPressMV		: REAL;	//Messspannung bei "rMinPress" in V
	rMaxPressMV		: REAL;	//Messspannung bei "rMaxPress" in V
	rFactorSetPress	: REAL := 1.0; //Faktor für Solldruck
	rFactorCurrPress: REAL:= 1.0; //Faktor für Istdruck	
	nOffsetSetPress	: INT;	//Offset für Solldruck
	nOffsetCurrPress: INT;	//Offset für Istdruck
END_VAR

VAR_STAT
	nHighestChannel : USINT;
END_VAR

nCurrentPress := REAL_TO_INT(F_YFuncX(rxMin:= rMinPressMV,
							rxMax:= rMaxPressMV,
							ryMin:= rMinPress,
							ryMax:= rMaxPress,
							rx:= 10.0 / 32767.0 * nAnalogInput)* rFactorCurrPress) + nOffsetCurrPress;

METHOD FB_init : BOOL
VAR_INPUT
	bInitRetains : BOOL; // if TRUE, the retain variables are initialized (warm start / cold start)
	bInCopyCode : BOOL;  // if TRUE, the instance afterwards gets moved into the copy code (online change)
END_VAR
nHighestChannel := nHighestChannel + 1;
nChannel := nHighestChannel;
END_METHOD

METHOD M_GetPressOk : BOOL
VAR_INPUT
	nSetPressure	: INT;
	nTolerancePlus	: INT;
	nToleranceMinus	: INT;
END_VAR
nCurrentPress := P_nCurrentPressure;
M_GetPressOk := (nCurrentPress >= nSetPressure - nToleranceMinus) AND (nCurrentPress <= nSetPressure + nTolerancePlus);
END_METHOD

METHOD M_SetPressure : ERRORID
VAR_INPUT
	nPressure		: INT;
END_VAR

VAR
	rAnaOut			: REAL;
END_VAR
//Solldruck muss zwischen min und max liegen oder 0
IF nPressure >= rMinPress OR nPressure <= rMaxPress OR nPressure = 0 THEN
	nSetPress := REAL_TO_INT(nPressure * rFactorSetPress);
	nSetPress := nPressure + nOffsetSetPress;
		 
	rAnaOut := F_YFuncX(rxMin:= rMinPress,
						rxMax:= rMaxPress,
						ryMin:= rMinPressCV,
						ryMax:= rMaxPressCV,
						rx:= nSetPress) * 32767.0 / 10.0;
	
	IF nPressure <> 0 THEN
		nAnalogOutput := REAL_TO_INT(rAnaOut);
		bSupplyActor := TRUE;
	ELSE
		nAnalogOutput := 0;
		bSupplyActor := FALSE;
	END_IF
ELSE
	M_SetPressure := E_ErrorIdCmd.ERRORID_InvalidPressure;
END_IF
END_METHOD

PROPERTY P_bSupplyOk : BOOL
GET
IF rMaxPress <= 0 THEN
	P_bSupplyOk := NOT bSupplyOk;
ELSE
	P_bSupplyOk := bSupplyOk;
END_IF
END_GET
END_PROPERTY

PROPERTY P_nCurrentPressure : INT
GET
P_nCurrentPressure := nCurrentPress;
END_GET
END_PROPERTY

PROPERTY P_nFactCurrPress : DINT
GET
P_nFactCurrPress := REAL_TO_DINT(rFactorCurrPress * 1000000.0);
END_GET
SET
rFactorCurrPress := DINT_TO_REAL(P_nFactCurrPress) / 1000000.0;
fbSettings.M_WritePersData();
END_SET
END_PROPERTY

PROPERTY P_nFactSetPress : DINT
GET
P_nFactSetPress := REAL_TO_DINT(rFactorSetPress * 1000000.0);
END_GET
SET
rFactorSetPress := DINT_TO_REAL(P_nFactSetPress) / 1000000.0;
fbSettings.M_WritePersData();
END_SET
END_PROPERTY

PROPERTY P_nMaxPress : DINT
GET
P_nMaxPress := REAL_TO_DINT(rMaxPress);
END_GET
SET
 rMaxPress := DINT_TO_REAL(P_nMaxPress);
 fbSettings.M_WritePersData();
END_SET
END_PROPERTY

PROPERTY P_nMaxPressCV : DINT
GET
P_nMaxPressCV := REAL_TO_DINT(rMaxPressCV * 1000);
END_GET
SET
rMaxPressCV := DINT_TO_REAL(P_nMaxPressCV) / 1000;
fbSettings.M_WritePersData();
END_SET
END_PROPERTY

PROPERTY P_nMaxPressMV : DINT
GET
P_nMaxPressMV := REAL_TO_DINT(rMaxPressMV * 1000);
END_GET
SET
rMaxPressMV := DINT_TO_REAL(P_nMaxPressMV) / 1000;
fbSettings.M_WritePersData();
END_SET
END_PROPERTY

PROPERTY P_nMinPress : DINT
GET
P_nMinPress := REAL_TO_DINT(rMinPress);
END_GET
SET
rMinPress := DINT_TO_REAL(P_nMinPress);
fbSettings.M_WritePersData();
END_SET
END_PROPERTY

PROPERTY P_nMinPressCV : DINT
GET
P_nMinPressCV := REAL_TO_DINT(rMinPressCV * 1000);
END_GET
SET
rMinPressCV := DINT_TO_REAL(P_nMinPressCV) / 1000;
fbSettings.M_WritePersData();
END_SET
END_PROPERTY

PROPERTY P_nMinPressMV : DINT
GET
P_nMinPressMV := REAL_TO_DINT(rMinPressMV * 1000);
END_GET
SET
rMinPressMV := DINT_TO_REAL(P_nMinPressMV) / 1000;
fbSettings.M_WritePersData();
END_SET
END_PROPERTY

PROPERTY P_nOffsetCurrPress : DINT
GET
P_nOffsetCurrPress := nOffsetCurrPress;
END_GET
SET
nOffsetCurrPress := DINT_TO_INT(P_nOffsetCurrPress);
END_SET
END_PROPERTY

PROPERTY P_nOffsetSetPress : DINT
GET
P_nOffsetSetPress := nOffsetSetPress;
END_GET
SET
nOffsetSetPress := DINT_TO_INT(P_nOffsetSetPress);
END_SET
END_PROPERTY

PROPERTY P_nSetPressure : INT
GET
P_nSetPressure := nSetPress;
END_GET
END_PROPERTY

END_FUNCTION_BLOCK

// ---- Hardware/FBox/PneuChannels/FB_SetPressure.TcPOU
FUNCTION_BLOCK FB_SetPressure
VAR_INPUT
	bExecute 		: BOOL;
	nValue			: INT;
	bAwait			: BOOL;	//Baustein bleibt solange busy, bis sich Solldruck in Toleranzfester eingestellt hat.
	tTimeout		: TIME;
	nTolerancePlus	: INT;
	nToleranceMinus	: INT;
END_VAR
VAR_OUTPUT
	bBusy : BOOL;
	bError : BOOL;
	nErrorId : ERRORID;		
END_VAR
VAR_IN_OUT
	pPneuChannelRef : POINTER TO FB_PneuChannelRef;
END_VAR
VAR
	nState : USINT;
	timer : TON;
END_VAR

IF bExecute THEN
	IF pPneuChannelRef = 0 THEN
		bBusy := FALSE;
		bError := TRUE;
		nErrorId := E_ErrorIdObjMgmt.ERRORID_InvalidHardwareRef;
		nState := 99;
		RETURN;
	END_IF
	
	IF nState = 0 THEN
		nErrorId := pPneuChannelRef^.M_SetPressure(nValue);
		IF nErrorId > 0 THEN
			bError := TRUE;
			RETURN;
		END_IF
		
		IF NOT bAwait THEN
			RETURN;
		END_IF
		nState := 1;
	END_IF
	
	IF nState = 1 THEN
		bBusy := TRUE;
		//falls Druck schon im Tolerenzbereich liegt, dann kann der FB sofort beendet werden
		IF pPneuChannelRef^.M_GetPressOk(nSetPressure:= nValue, nTolerancePlus:= nTolerancePlus, nToleranceMinus:= nToleranceMinus) THEN
			bBusy := FALSE;
			nState := 2;
			RETURN;
		END_IF
		
		//Timer für Timout starten
		timer(IN:= TRUE, PT:= tTimeout);
		IF timer.Q THEN
			bBusy := FALSE;
			bError := TRUE;
			nErrorId := E_ErrorIdCmd.ERRORID_PressTimeOut;
			nState := 99;
			RETURN;
		END_IF
	END_IF
	
ELSE
	nState := 0;
	bBusy := FALSE;
	bError := FALSE;
	nErrorId := 0;
	timer(IN:=FALSE);
END_IF

END_FUNCTION_BLOCK

// ---- Objects/Tools/FB_Exposure.TcPOU
FUNCTION_BLOCK FB_Exposure EXTENDS FB_GCodeTool
VAR_INPUT
END_VAR
VAR_OUTPUT
	
END_VAR
VAR
	//Reference zu TripleTrigger
	pTripleTrigRef : POINTER TO FB_HwRefTripleTrigger;

	//Specproperties
	rWorkingDistance		: REAL;
	bInvertWorkingDistance 	: BOOL;
	eTriggerType			: E_TriggerOutput;
	nTriggerBehavior		: USINT;
	nTriggerChannel			: USINT;
	
	//****************************************Aktionvariablen****************************************************
	stActionDataSpec	: ST_ActionData;
	
	//Action: "InitTool"
	bInitTool			: BOOL;
	nStateA_InitTool	: USINT;
	
	//Action: "Expose"
	bExpose				: BOOL;
	nStateA_Expose		: USINT;
	nBrightness			: UINT;
	bExposeStart		: BOOL;
	timer				: TON;
	bSecondCycle		: BOOL;
	nCycleCnt			: USINT;
END_VAR

IF eCurrentState = E_MachineState.MACHINESTATE_Active THEN
	IF bInitTool THEN
		A_InitTool();
		IF nStateA_InitTool >= 80 THEN
			IF nStateA_InitTool >= 99 THEN
				bError := TRUE;		
			END_IF
			bInitTool := FALSE;
			nStateA_InitTool := 0;
			M_RemoveListEntry(nSearchValue:= E_Action.ACTION_Init);
		END_IF		
	END_IF

	IF bExpose THEN
		A_Expose();
		IF nStateA_Expose >= 80 THEN
			IF nStateA_Expose >= 99 THEN
				bError := TRUE;	
			END_IF
			bExpose := FALSE;
			nStateA_Expose := 0;
			M_RemoveListEntry(nSearchValue:= E_Action.ACTION_Expose);
		END_IF
	END_IF
END_IF

//FB_MzTool aufrufen
SUPER^();

//Prozessdaten aktualisieren
CASE eTriggerType OF
	E_TriggerOutput.PlcOutput:
		stProcessData.n32Data[7] := BOOL_TO_DINT(fbPlcTriggerOut.M_GetState(nTriggerChannel));
	E_TriggerOutput.MultiZOutput:
		stProcessData.n32Data[7] := BOOL_TO_DINT(fbMultiZDigiOut.M_GetState(nTriggerChannel));
	E_TriggerOutput.MultiZPWM:
		stProcessData.n32Data[7] := BOOL_TO_DINT(fbMultiZPWM.M_GetState(nTriggerChannel));
	E_TriggerOutput.TripleTriggerModul:
		stProcessData.n32Data[7] := BOOL_TO_DINT(pTripleTrigRef^.M_GetState(nTriggerChannel));
END_CASE

aObjProcData[nNotifyId] := stProcessData;

ACTION A_Expose:
CASE nStateA_Expose OF
	0:	
		CASE eTriggerType OF
			E_TriggerOutput.PlcOutput:
				fbPlcTriggerOut.M_On(nTriggerChannel); //muss in jedem Zylus neu aufgerufen werden (aus Sicherheitsgründen)
			E_TriggerOutput.MultiZOutput:
				fbMultiZDigiOut.M_On(nTriggerChannel); //muss in jedem Zylus neu aufgerufen werden (aus Sicherheitsgründen)
			E_TriggerOutput.MultiZPWM:
				fbMultiZPWM.M_On(nTriggerChannel,1000); //muss in jedem Zylus neu aufgerufen werden (aus Sicherheitsgründen) (100% Tastverhältnis)
			E_TriggerOutput.TripleTriggerModul:
				pTripleTrigRef^.M_SetAmplitudePercent(nTriggerChannel,nBrightness);//Helligkeit
				pTripleTrigRef^.M_SetPulse(nTriggerChannel,65535); //Dauersignal
				pTripleTrigRef^.M_TriggerOn(nTriggerChannel,0);
		END_CASE	

		//Timer starten
		IF timer.PT > T#0S THEN
			timer(IN:=TRUE);
		END_IF
		bSecondCycle := FALSE;
		nCycleCnt := 0;
		nStateA_Expose := 1;
		
	1:	//Warten, bis Zeit abgelaufen oder TriggerState  = FALSE
		timer();
		IF timer.Q THEN
			timer(IN:= FALSE);
			CASE eTriggerType OF
				E_TriggerOutput.PlcOutput:
					fbPlcTriggerOut.M_Off(nTriggerChannel);
				E_TriggerOutput.MultiZOutput:
					fbMultiZDigiOut.M_Off(nTriggerChannel);
				E_TriggerOutput.MultiZPWM:
					fbMultiZPWM.M_Off(nTriggerChannel);
				E_TriggerOutput.TripleTriggerModul:
					pTripleTrigRef^.M_TriggerOff(nTriggerChannel);
			END_CASE
		END_IF
		
		CASE eTriggerType OF
			E_TriggerOutput.PlcOutput:
				IF NOT fbPlcTriggerOut.M_GetState(nTriggerChannel) THEN
					nStateA_Expose := 2;
				ELSE
					fbPlcTriggerOut.M_On(nTriggerChannel);
				END_IF
			E_TriggerOutput.MultiZOutput:
				IF NOT fbMultiZDigiOut.M_GetState(nTriggerChannel) THEN
					nStateA_Expose := 80;
				ELSE
					fbMultiZDigiOut.M_On(nTriggerChannel);
				END_IF
			E_TriggerOutput.MultiZPWM:
				IF NOT fbMultiZPWM.M_GetState(nTriggerChannel) THEN
					nStateA_Expose := 80;
				ELSE
					fbMultiZPWM.M_On(nTriggerChannel, 1000);
				END_IF
			E_TriggerOutput.TripleTriggerModul:
				nCycleCnt := nCycleCnt + 1;
				IF nCycleCnt = 2 THEN
					IF NOT pTripleTrigRef^.M_GetState(nTriggerChannel) THEN
						timer(IN:= FALSE);
						pTripleTrigRef^.M_TriggerOff(nTriggerChannel);
						nStateA_Expose := 2;
					END_IF
				END_IF
		END_CASE

	2:	//Delay bis ready (Blendenschaltzeit) (für Omnicure)
		timer(IN:=TRUE,PT:=T#500MS);
		IF timer.Q THEN
			timer(IN:=FALSE);
			nStateA_Expose := 80;
		END_IF
		
	70:	//Abbrechen
		timer(IN:= FALSE);
		CASE eTriggerType OF
			E_TriggerOutput.PlcOutput:
				fbPlcTriggerOut.M_Off(nTriggerChannel);
			E_TriggerOutput.MultiZOutput:
				fbMultiZDigiOut.M_Off(nTriggerChannel);
			E_TriggerOutput.MultiZPWM:
				fbMultiZPWM.M_Off(nTriggerChannel);
			E_TriggerOutput.TripleTriggerModul:
				pTripleTrigRef^.M_TriggerOff(nTriggerChannel);
		END_CASE
		nStateA_Expose := 80;
END_CASE
END_ACTION

ACTION A_InitTool:
nStateA_InitTool := 80;
END_ACTION

ACTION A_Reset:
//Ist noch eine Aktion aktiv?
IF nStateA_ResetSpec = 0 THEN 
	IF bExpose THEN
		bExpose := FALSE;
		nStateA_Expose := 0;
	END_IF
	
	nStateA_ResetSpec := 80;
END_IF

SUPER^.A_Reset();
END_ACTION

ACTION A_Stop:
IF nStateA_Stop = 0 THEN

	IF bExpose AND nStateA_Expose < 70 THEN
		nStateA_Expose := 70;
	END_IF
	
	nStateA_Stop := 1;
END_IF

SUPER^.A_Stop();
END_ACTION

METHOD FB_init : BOOL
VAR_INPUT
	bInitRetains : BOOL; // if TRUE, the retain variables are initialized (warm start / cold start)
	bInCopyCode : BOOL;  // if TRUE, the instance afterwards gets moved into the copy code (online change)
END_VAR
eObjectType := E_ObjectType.OBJECTTYPE_Exposure;
eObjectGroup := E_ObjectGroup.OBJECTGROUP_MzTool OR E_ObjectGroup.OBJECTGROUP_Device;
END_METHOD

METHOD M_AddChild : ERRORID
VAR_INPUT
	pObject : POINTER TO FB_Object;
	nSlotNr	: UINT;
	nIndex 	: INT;
END_VAR
//Der Exoser kann folgende Objekt-Typen aufnehmen
//Camera, Exposure
IF pObject > 0 THEN
	IF pObject^.P_eObjectType = E_ObjectType.OBJECTTYPE_Camera OR
		pObject^.P_eObjectType = E_ObjectType.OBJECTTYPE_DummyTool OR
		pObject^.P_eObjectType = E_ObjectType.OBJECTTYPE_Exposure THEN
		
		M_AddChild := SUPER^.M_AddChild(pObject,nSlotNr,nIndex);
	ELSE
		M_AddChild := E_ErrorIdObjMgmt.ERRORID_InvalidParentObject;
	END_IF
ELSE
	M_AddChild := E_ErrorIdObjMgmt.ERRORID_InvalidParentObject;
END_IF
END_METHOD

METHOD M_CancelAction
VAR_INPUT
	eAction : E_Action;
END_VAR
IF eAction = E_Action.ACTION_Expose THEN
	IF bExpose AND nStateA_Expose < 70 THEN
		nStateA_Expose := 70;
	END_IF
ELSE
	SUPER^.M_CancelAction(eAction);
END_IF
END_METHOD

METHOD M_CheckAction : ERRORID
VAR_INPUT
	refActionData 	: REFERENCE TO ST_ActionData;
	pCorrelObject	: POINTER TO FB_Object;
END_VAR
CASE refActionData.eAction OF
	E_Action.ACTION_Expose: //BasicAction für ActionOnArray
ELSE
	M_CheckAction := SUPER^.M_CheckAction(refActionData, pCorrelObject);
END_CASE
END_METHOD

METHOD M_CheckProps : ERRORID
VAR_INPUT
END_VAR
M_CheckProps := SUPER^.M_CheckProps();
IF M_CheckProps > 0 THEN
	RETURN;
END_IF

IF eTriggerType = E_TriggerOutput.TripleTriggerModul AND pTripleTrigRef = 0 THEN
	M_CheckProps := E_ErrorIdObjMgmt.ERRORID_InvalidHardwareRef;
END_IF
END_METHOD

METHOD M_ExeAction : ERRORID
VAR_INPUT
	refActionData : REFERENCE TO ST_ActionData;	
END_VAR
IF NOT (eCurrentState = E_MachineState.MACHINESTATE_Idle OR
	eCurrentState = E_MachineState.MACHINESTATE_Active OR
	eCurrentState = E_MachineState.MACHINESTATE_Ready) THEN
	M_ExeAction := E_ErrorIdCmd.ERRORID_InvalidState;
	RETURN;
END_IF

CASE refActionData.eAction OF
	
	E_Action.ACTION_Init:
		IF NOT bInitAxis AND NOT bInitTool THEN
			bInitAxis := TRUE;
			bInitTool := TRUE;
			fbList.A_AddHeadValue( hList := hList, putValue := E_Action.ACTION_Init);	//InitAxis
			fbList.A_AddHeadValue( hList := hList, putValue := E_Action.ACTION_Init);	//InitTool
		ELSE
			RETURN;
		END_IF
		
	E_Action.ACTION_Expose:
		bExposeStart := DINT_TO_BOOL(refActionData.aParams[1]);
		IF NOT bExpose AND bExposeStart THEN
			nBrightness := DINT_TO_UINT(refActionData.aParams[2]);
			timer.PT := DINT_TO_TIME(refActionData.aParams[3]);
			fbList.A_AddHeadValue( hList := hList, putValue := E_Action.ACTION_Expose);
			bExpose := TRUE;
		ELSIF NOT bExposeStart THEN
			CASE eTriggerType OF
				E_TriggerOutput.PlcOutput:
					fbPlcTriggerOut.M_Off(nTriggerChannel);
				E_TriggerOutput.TripleTriggerModul:
					pTripleTrigRef^.M_TriggerOff(nTriggerChannel);
				E_TriggerOutput.MultiZOutput:
					fbMultiZDigiOut.M_Off(nTriggerChannel);
				E_TriggerOutput.MultiZPWM:
					fbMultiZPWM.M_Off(nTriggerChannel);
			END_CASE
		ELSE
			RETURN;	
		END_IF
	ELSE
		M_ExeAction := SUPER^.M_ExeAction(refActionData);
		RETURN;
END_CASE
bBusy := TRUE;
eCurrentState := E_MachineState.MACHINESTATE_Active;
END_METHOD

METHOD M_GetAllProps : ERRORID
VAR_INPUT
	refCmdData : REFERENCE TO  ST_CmdData;
END_VAR
SUPER^.M_GetAllProps(refCmdData);
nCurrentPropIndex := nCurrentPropIndex + 1;
refCmdData.n32Data[nCurrentPropIndex] := REAL_TO_DINT(rWorkingDistance);
nCurrentPropIndex := nCurrentPropIndex + 1;
refCmdData.n32Data[nCurrentPropIndex] := BOOL_TO_DINT(bInvertWorkingDistance);
nCurrentPropIndex := nCurrentPropIndex + 1;
refCmdData.n32Data[nCurrentPropIndex] := eTriggerType;
nCurrentPropIndex := nCurrentPropIndex + 1;
refCmdData.n32Data[nCurrentPropIndex] := nTriggerBehavior;
nCurrentPropIndex := nCurrentPropIndex + 1;
refCmdData.n32Data[nCurrentPropIndex] := nTriggerChannel;
END_METHOD

METHOD M_SetAllProps : ERRORID
VAR_INPUT
	refCmdData : REFERENCE TO  ST_CmdData;
END_VAR
M_SetAllProps := SUPER^.M_SetAllProps(refCmdData);

IF M_SetAllProps > 0 THEN
	RETURN;
END_IF

//WorkingDistance
nCurrentPropIndex := nCurrentPropIndex + 1;
nSpecPropIndex := nCurrentPropIndex;
rWorkingDistance := DINT_TO_REAL(refCmdData.n32Data[nCurrentPropIndex]);
nCurrentPropIndex := nCurrentPropIndex + 1;
bInvertWorkingDistance := DINT_TO_BOOL(refCmdData.n32Data[nCurrentPropIndex]);

//TriggerType
nCurrentPropIndex := nCurrentPropIndex + 1;
eTriggerType := DINT_TO_USINT(refCmdData.n32Data[nCurrentPropIndex]);
pTripleTrigRef := 0;

//TriggerBehavior
nCurrentPropIndex := nCurrentPropIndex + 1;
nTriggerBehavior := DINT_TO_USINT(refCmdData.n32Data[nCurrentPropIndex]);
IF NOT (nTriggerBehavior >= 0 AND nTriggerBehavior <= 1) THEN
	M_SetAllProps := E_ErrorIdObjMgmt.ERRORID_InvalidTriggerChannel;
	RETURN;
END_IF

//TriggerChannel
nCurrentPropIndex := nCurrentPropIndex + 1;
nTriggerChannel := DINT_TO_USINT(refCmdData.n32Data[nCurrentPropIndex]);

CASE eTriggerType OF
	E_TriggerOutput.PlcOutput,
	E_TriggerOutput.MultiZOutput:
		IF NOT (nTriggerChannel >= 1 AND nTriggerChannel <= 3) THEN
			M_SetAllProps := E_ErrorIdObjMgmt.ERRORID_InvalidTriggerChannel;
			RETURN;
		END_IF
	E_TriggerOutput.MultiZPWM:
		IF NOT (nTriggerChannel >= 1 AND nTriggerChannel <= 2) THEN
			M_SetAllProps := E_ErrorIdObjMgmt.ERRORID_InvalidTriggerChannel;
			RETURN;
		END_IF	
	E_TriggerOutput.TripleTriggerModul:
		{IF defined (variable:aFbTripleTriggerRef)}
		IF NOT (nTriggerChannel >= 1 AND nTriggerChannel <= 3) THEN
			M_SetAllProps := E_ErrorIdObjMgmt.ERRORID_InvalidTriggerChannel;
		END_IF
		pTripleTrigRef := ADR(aFbTripleTriggerRef[1]);
		{ELSE}
		M_SetAllProps := E_ErrorIdObjMgmt.ERRORID_InvalidHardwareRef;
		RETURN;
		{END_IF}	
END_CASE

nNoOfProps := nCurrentPropIndex + 1;
END_METHOD

METHOD M_SetSingleProp : ERRORID
VAR_INPUT
	refCmdData : REFERENCE TO  ST_CmdData;
END_VAR

VAR
	nTriggerChannel : USINT;
END_VAR
IF nSpecPropIndex = refCmdData.aHeader[1] THEN
	rWorkingDistance := DINT_TO_REAL(refCmdData.n32Data[0]);
ELSIF nSpecPropIndex + 1 = refCmdData.aHeader[1] THEN
	bInvertWorkingDistance := DINT_TO_BOOL(refCmdData.n32Data[0]);
ELSIF nSpecPropIndex + 4 = refCmdData.aHeader[1] THEN
	nTriggerChannel := DINT_TO_USINT(refCmdData.n32Data[0]);
	IF eTriggerType = E_TriggerOutput.MultiZPWM THEN
		IF NOT (nTriggerChannel >= 1 AND nTriggerChannel <= 2) THEN
			M_SetSingleProp := E_ErrorIdObjMgmt.ERRORID_InvalidTriggerChannel;
			RETURN;
		END_IF
		THIS^.nTriggerChannel := nTriggerChannel;
	ELSE
		IF NOT (nTriggerChannel >= 1 AND nTriggerChannel <= 3) THEN
			M_SetSingleProp := E_ErrorIdObjMgmt.ERRORID_InvalidTriggerChannel;
			RETURN;
		END_IF
		THIS^.nTriggerChannel := nTriggerChannel;
	END_IF
ELSE
	M_SetSingleProp := SUPER^.M_SetSingleProp(refCmdData);
END_IF
END_METHOD

PROPERTY P_stAbsPosTotal : ST_3DPoint
GET
VAR
	stPosTemp : ST_3DPoint;
END_VAR
stPosTemp := SUPER^.P_stAbsPosPhys;
IF bInvertWorkingDistance THEN
	stPosTemp.Z := stPosTemp.Z + rWorkingDistance;
ELSE
	stPosTemp.Z := stPosTemp.Z - rWorkingDistance;
END_IF
P_stAbsPosTotal := stPosTemp;
END_GET
END_PROPERTY

PROPERTY P_stCurrentPosTotal : ST_3DPoint
GET
VAR
	stPosTemp : ST_3DPoint;
END_VAR
stPosTemp := P_stCurrentPosPhys;
IF bInvertWorkingDistance THEN
	stPosTemp.Z := stPosTemp.Z + rWorkingDistance;
ELSE
	stPosTemp.Z := stPosTemp.Z - rWorkingDistance;
END_IF
P_stCurrentPosTotal := stPosTemp;
END_GET
END_PROPERTY

END_FUNCTION_BLOCK

// ---- Hardware/FBox/FB_HwRefTripleTrigger.TcPOU
FUNCTION_BLOCK FB_HwRefTripleTrigger EXTENDS FB_CanNodeBase
VAR_INPUT
END_VAR
VAR_OUTPUT
END_VAR
VAR
	//PDOs
	nState 			AT %I* : ARRAY[1..3] OF USINT;
	nError 			AT %I* : USINT;
	nPeriod 		AT %Q* : ARRAY[1..3] OF UINT;
	nPulse 			AT %Q* : ARRAY[1..3] OF UINT;
	nPulseNumber 	AT %Q* : ARRAY[1..3] OF UINT;
	nVoltage 		AT %Q* : ARRAY[1..3] OF UINT;
	nCtrl 			AT %Q* : ARRAY[1..3] OF USINT;
	
	//SDOs
	nFrequency 			: ARRAY[1..3] OF DINT;
	nAmplitudePercent 	: ARRAY[1..3] OF UINT;
END_VAR

IF bNodeEnabled THEN
	SUPER^();
END_IF

METHOD M_SetPulse
VAR_INPUT
	nChannel : USINT;
	nPulse : UINT;
END_VAR
THIS^.nPulse[nChannel] := nPulse;
END_METHOD

METHOD M_SetFrequency
VAR_INPUT
	nChannel : USINT;
	nFrequency : DINT;
END_VAR
IF nFrequency > 0 THEN
	THIS^.nFrequency[nChannel] := nFrequency;
	nPeriod[nChannel] := DINT_TO_UINT(1000000 / nFrequency);
ELSE
	nPeriod[nChannel] := 0;
	THIS^.nFrequency[nChannel] := 0;
END_IF
END_METHOD

METHOD M_TriggerOn
VAR_INPUT
	nChannel : USINT;
	nPulseNumber : UINT;
END_VAR
THIS^.nPulseNumber[nChannel] := nPulseNumber;
nCtrl[nChannel] := 1;
END_METHOD

METHOD M_GetAmlitudeVolt : UINT
VAR_INPUT
	nChannel : USINT;
END_VAR
M_GetAmlitudeVolt := nVoltage[nChannel];
END_METHOD

METHOD M_TriggerOff
VAR_INPUT
	nChannel : USINT;
END_VAR
nCtrl[nChannel] := 0;
END_METHOD

METHOD M_GetState : BOOL
VAR_INPUT
	nChannel : USINT;
END_VAR
M_GetState := nState[nChannel].0;
END_METHOD

METHOD M_GetPulse : UINT
VAR_INPUT
	nChannel : USINT;
END_VAR
M_GetPulse := nPulse[nChannel];
END_METHOD

METHOD M_GetAmplitudePercent : UINT
VAR_INPUT
	nChannel : USINT;
END_VAR
M_GetAmplitudePercent := nAmplitudePercent[nChannel];
END_METHOD

METHOD M_SetAmplitudeVolt
VAR_INPUT
	nChannel : USINT;
	nValue : UINT;
END_VAR
nVoltage[nChannel] := LIMIT(0,nValue,10000);
nAmplitudePercent[nChannel] := nVoltage[nChannel] * 1000 / 10000;
END_METHOD

METHOD M_SetAmplitudePercent
VAR_INPUT
	nChannel : USINT;
	nValue : UINT;	//Zehntel %
END_VAR
nAmplitudePercent[nChannel] := LIMIT(0,nValue,1000);
nVoltage[nChannel] := 10000 / 1000 * nAmplitudePercent[nChannel];
END_METHOD

METHOD M_GetFrequency : DINT
VAR_INPUT
	nChannel : USINT;
END_VAR
M_GetFrequency := nFrequency[nChannel];
END_METHOD

END_FUNCTION_BLOCK

// ---- Objects/Tools/FB_HybridDispenser.TcPOU
FUNCTION_BLOCK FB_HybridDispenser EXTENDS FB_GCodeTool IMPLEMENTS I_Dispenser
VAR_INPUT
END_VAR
VAR_OUTPUT
END_VAR
VAR
	//Specproperties
	aiDispenser		: ARRAY[1..3] OF I_Dispenser;
	nMasterSlotNr	: USINT;

	//****************************************Aktionsvariablen****************************************************
	bBasicDispense			: BOOL;
	nStateA_BasicDispense 	: USINT;
	
	n : INT; //Zählvariablen
	m : INT; //Zählvariablen

END_VAR

IF eCurrentState = E_MachineState.MACHINESTATE_Active THEN
	IF bBasicDispense THEN
		A_HybridDispense();
		IF nStateA_BasicDispense >= 80 THEN
			IF nStateA_BasicDispense >= 99 THEN
				bError := TRUE;
			END_IF
			bBasicDispense := FALSE;
			nStateA_BasicDispense := 0;
			M_RemoveListEntry(nSearchValue:= E_Action.ACTION_BasicDispense);
		END_IF
	END_IF
END_IF

SUPER^();	//FB_MzTool aufrufen

//Prozessdaten aktualisieren
stProcessData.n32Data[7] := BOOL_TO_DINT(bBasicDispense);
aObjProcData[nNotifyId] := stProcessData;

ACTION A_HybridDispense:
IF nStateA_BasicDispense = 0 THEN	//alle Dispenser starten
	FOR n := 1 TO 3 BY 1 DO
		IF aiDispenser[n] <> 0 THEN
			stError.ErrorId := aiDispenser[n].M_DispenserStart();
			stError.ObjectId := aiDispenser[n].P_pObject^.P_nObjectID;
			IF stError.ErrorId > 0 THEN
				//Bereits gestartete Tools wieder stoppen
				FOR m := 1 TO n - 1 BY 1 DO
					aiDispenser[m].M_DispenserStop();
				END_FOR
				nStateA_BasicDispense := 99;
				EXIT;
			END_IF
		END_IF
	END_FOR
	IF nStateA_BasicDispense = 0 THEN
		nStateA_BasicDispense := 1;	
	END_IF
END_IF

IF nStateA_BasicDispense = 1 THEN	//alle Dispenser laufen -> permanent auf Fehler überwachen
	//Das Verlassen dieses States erfolgt durch die Action "HybridDispense" mit Parameter "off" oder durch Stop bzw. Cancel
	FOR n := 1 TO 3 BY 1 DO
		IF aiDispenser[n] <> 0 THEN
			IF aiDispenser[n].P_bError THEN
				stError.ErrorId := aiDispenser[n].P_nErrorId;
				stError.ObjectId := aiDispenser[n].P_pObject^.P_nObjectID;
				nStateA_BasicDispense := 2; //weiter zu stoppen
				EXIT;
			END_IF
		END_IF
	END_FOR	
END_IF

IF nStateA_BasicDispense = 2 THEN //übrige Dispenser nach Fehler stoppen
	nStateA_BasicDispense := 99;
	FOR n := 1 TO 3 BY 1 DO
		IF aiDispenser[n] <> 0 THEN
			IF NOT aiDispenser[n].P_bError THEN
				aiDispenser[n].M_DispenserStop();
			END_IF
		END_IF
	END_FOR	
END_IF

IF nStateA_BasicDispense = 70 THEN //Dispenser stoppen
	nStateA_BasicDispense := 71;
	FOR n := 1 TO 3 BY 1 DO
		IF aiDispenser[n] <> 0 THEN
			aiDispenser[n].M_DispenserStop();
		END_IF
	END_FOR	
ELSIF nStateA_BasicDispense = 71 THEN //warten bis alle Dispenser gestoppt
	nStateA_BasicDispense := 80;
	FOR n := 1 TO 3 BY 1 DO
		IF aiDispenser[n] <> 0 THEN
			IF NOT aiDispenser[n].P_eDispenserState = E_DispenserState.Idle THEN 
				nStateA_BasicDispense := 71;
			END_IF
		END_IF
	END_FOR	
END_IF

//Errorhandling
IF nStateA_BasicDispense = 99 THEN
	stError.Cmd := E_Action.ACTION_BasicDispense;
	stError.POU := E_POU.POU_FB_HybridDispenser;
	stError.POUAction := E_POUACT.POUACT_A_BasicDispense;
	fbErrorList.M_Add(stError);
END_IF
END_ACTION

ACTION A_Reset:
//Ist noch eine Aktion aktiv?
IF nStateA_ResetSpec = 0 THEN 
	(*IF bHeating THEN
		bHeating := FALSE;
		nStateA_Heating := 0;
	END_IF*)
	nStateA_ResetSpec := 80;
END_IF

SUPER^.A_Reset();
END_ACTION

ACTION A_Stop:
IF nStateA_Stop = 0 THEN
	IF bBasicDispense AND nStateA_BasicDispense = 1 THEN
		nStateA_BasicDispense := 70;
	END_IF
	nStateA_Stop := 1;	
END_IF

SUPER^.A_Stop();
END_ACTION

METHOD FB_init : BOOL
VAR_INPUT
	bInitRetains : BOOL; // if TRUE, the retain variables are initialized (warm start / cold start)
	bInCopyCode : BOOL;  // if TRUE, the instance afterwards gets moved into the copy code (online change)
END_VAR
eObjectType := E_ObjectType.OBJECTTYPE_HybridDispenser;
eObjectGroup := E_ObjectGroup.OBJECTGROUP_MzTool OR E_ObjectGroup.OBJECTGROUP_Device;
END_METHOD

METHOD M_AddChild : ERRORID
VAR_INPUT
	pObject : POINTER TO FB_Object;
	nSlotNr	: UINT;
	nIndex : INT;
END_VAR
//Der HybridDispenser kann folgende Objekttypen aufnehmen
//Extruder, PassivePip, CartDispenser
IF pObject > 0 THEN
	IF pObject^.P_eObjectType = E_ObjectType.OBJECTTYPE_Extruder OR
		pObject^.P_eObjectType = E_ObjectType.OBJECTTYPE_CartDispenser OR
		pObject^.P_eObjectType = E_ObjectType.OBJECTTYPE_CartDispStirrer OR
		pObject^.P_eObjectType = E_ObjectType.OBJECTTYPE_PassivPip THEN
		M_AddChild := SUPER^.M_AddChild(pObject,nSlotNr,nIndex);
	ELSE
		M_AddChild := E_ErrorIdObjMgmt.ERRORID_InvalidParentObject;
	END_IF
ELSE
	M_AddChild := E_ErrorIdObjMgmt.ERRORID_InvalidParentObject;
END_IF
END_METHOD

METHOD M_CancelAction
VAR_INPUT
	eAction : E_Action;
END_VAR
CASE eAction OF
	E_Action.ACTION_BasicDispense:
		IF bBasicDispense AND nStateA_BasicDispense = 1 THEN
			nStateA_BasicDispense := 70;
		END_IF
ELSE
	SUPER^.M_CancelAction(eAction);
END_CASE
END_METHOD

METHOD M_CheckAction : ERRORID
VAR_INPUT
	refActionData 	: REFERENCE TO ST_ActionData;
	pCorrelObject	: POINTER TO FB_Object;
END_VAR
CASE refActionData.eAction OF
	E_Action.ACTION_Dispense,
	E_Action.ACTION_CleanTip,
	E_Action.ACTION_MeasureTool,
	E_Action.ACTION_TeachTarget:
		RETURN;
ELSE
	M_CheckAction := SUPER^.M_CheckAction(refActionData, pCorrelObject);
END_CASE
END_METHOD

METHOD M_CheckGCodeStart : ERRORID
VAR_INPUT
END_VAR

VAR
	i : USINT;
	pGCodeTool : POINTER TO FB_GCodeTool;
END_VAR
FOR i := 1 TO 3 BY 1 DO
	IF aiDispenser[i] <> 0 AND_THEN aiDispenser[i].P_pObject^.P_eObjectType = E_ObjectType.OBJECTTYPE_Extruder THEN
		pGCodeTool := aiDispenser[i].P_pObject;
		M_CheckGCodeStart := pGCodeTool^.M_CheckGCodeStart();
		IF M_CheckGCodeStart > 0 THEN
			RETURN;
		END_IF
	END_IF
END_FOR
END_METHOD

METHOD M_CheckProcDataType : BOOL
VAR_INPUT
	eProcDataType : E_ProcDataType;
END_VAR
END_METHOD

METHOD M_CheckProps : ERRORID
VAR_INPUT
END_VAR

VAR
	i 				: UINT;
	pSlot 			: POINTER TO FB_Slot;
	pExtruder 		: POINTER TO FB_Extruder;
	pCartDispenser 	: POINTER TO FB_CartDispenser;
	pPassivePip 	: POINTER TO FB_PassivPip;
END_VAR
M_CheckProps := SUPER^.M_CheckProps();
//Kann bis zu 3 CartDispenser enthalten
aiDispenser[1] := 0;
aiDispenser[2] := 0;
aiDispenser[3] := 0;
FOR i:= 1 TO nNumberOfSlots BY 1 DO
	pSlot := fbSlotList.M_GetAtNr(i);
	IF pSlot > 0 AND_THEN pSlot^.P_pChild > 0  THEN
		//Achtung, nur Tools die das Interface "I_HybridDispenser" implementieren sind erlaubt!
		IF pSlot^.P_pChild^.P_eObjectType = E_ObjectType.OBJECTTYPE_Extruder THEN
			pExtruder := pSlot^.P_pChild;
			aiDispenser[pSlot^.P_nNr] := pExtruder^;
		ELSIF pSlot^.P_pChild^.P_eObjectType = E_ObjectType.OBJECTTYPE_CartDispenser OR 
				pSlot^.P_pChild^.P_eObjectType = E_ObjectType.OBJECTTYPE_CartDispStirrer THEN
			pCartDispenser := pSlot^.P_pChild;
			aiDispenser[pSlot^.P_nNr] := pCartDispenser^;
		ELSIF pSlot^.P_pChild^.P_eObjectType = E_ObjectType.OBJECTTYPE_PassivPip THEN
			pPassivePip := pSlot^.P_pChild;
			aiDispenser[pSlot^.P_nNr] := pPassivePip^;
		END_IF
	END_IF
END_FOR
//MasterSlotNr auswerten
//1. kann nur 1,2 oder 3 sein
//2. entsprechender Slot muss belegt sein
IF nMasterSlotNr >= 1 AND nMasterSlotNr <= 3 THEN
	IF aiDispenser[nMasterSlotNr] = 0 THEN
		M_CheckProps := E_ErrorIdObjMgmt.ERRORID_NoToolOnMasterSlot;	
	END_IF
ELSE
	M_CheckProps := E_ErrorIdObjMgmt.ERRORID_InvalidSlotNumber;
END_IF
END_METHOD

METHOD M_ClearAllProps
VAR_INPUT
	bIgnoreParent : BOOL; //Es wird das gesamte OD gelöscht. -> Zeiger auf Parent nicht mehr gültig!
END_VAR
aiDispenser[1] := 0;
aiDispenser[2] := 0;
aiDispenser[3] := 0;
SUPER^.M_ClearAllProps(bIgnoreParent);
END_METHOD

METHOD M_DispenserPrepare : ERRORID
VAR_INPUT
END_VAR
//do nothing
END_METHOD

METHOD M_DispenserStart : ERRORID
VAR_INPUT
END_VAR
IF NOT (eCurrentState = E_MachineState.MACHINESTATE_Idle OR
	eCurrentState = E_MachineState.MACHINESTATE_Active OR
	eCurrentState = E_MachineState.MACHINESTATE_Ready) THEN
	M_DispenserStart := E_ErrorIdCmd.ERRORID_InvalidState;
	RETURN;
END_IF
			
IF NOT bBasicDispense THEN
	bBasicDispense := TRUE;
	fbList.A_AddHeadValue(hList := hList, putValue := E_Action.ACTION_BasicDispense);
ELSE //Bereits Ein -> Error werfen
	M_DispenserStart := E_ErrorIdCmd.ERRORID_BasicActionActive;
	RETURN;
END_IF

bBusy := TRUE;
eCurrentState := E_MachineState.MACHINESTATE_Active;
END_METHOD

METHOD M_DispenserStop : ERRORID
VAR_INPUT
END_VAR
IF bBasicDispense AND nStateA_BasicDispense = 1 THEN
	nStateA_BasicDispense := 70;
END_IF
END_METHOD

METHOD M_ExeAction : ERRORID
VAR_INPUT
	refActionData : REFERENCE TO ST_ActionData;	
END_VAR
IF NOT (eCurrentState = E_MachineState.MACHINESTATE_Idle OR
	eCurrentState = E_MachineState.MACHINESTATE_Active OR
	eCurrentState = E_MachineState.MACHINESTATE_Ready) THEN
	M_ExeAction := E_ErrorIdCmd.ERRORID_InvalidState;
	RETURN;
END_IF

CASE refActionData.eAction OF
	E_Action.ACTION_BasicDispense:
		IF refActionData.aParams[1] = 0 THEN //Aus
			M_ExeAction := M_DispenserStop();
		ELSE //Ein
			M_ExeAction := M_DispenserStart();
		END_IF
	ELSE
		M_ExeAction := SUPER^.M_ExeAction(refActionData);
		RETURN;
END_CASE
END_METHOD

METHOD M_GetAllProps : ERRORID
VAR_INPUT
	refCmdData : REFERENCE TO  ST_CmdData;
END_VAR
SUPER^.M_GetAllProps(refCmdData);
nCurrentPropIndex := nCurrentPropIndex + 1;
refCmdData.n32Data[nCurrentPropIndex] := nMasterSlotNr;
END_METHOD

METHOD M_GetNozzle : POINTER TO FB_Nozzle
VAR_INPUT
END_VAR
IF P_pMasterTool > 0 THEN
	M_GetNozzle := P_pMasterTool^.M_GetNozzle();
END_IF
END_METHOD

METHOD M_GetProcData : DINT
VAR_INPUT
	eProcDataType : E_ProcDataType;
END_VAR
END_METHOD

METHOD M_GetZAxisRef : POINTER TO FB_ZAxisRef
VAR_INPUT
	pTool : POINTER TO FB_MzTool;
	pToolSlot : POINTER TO FB_Slot;
END_VAR

VAR
	nSlotDiff : INT;
	nAxisNr : INT;
END_VAR
//Diese Methode überschreibt sie Methode von FB_MzTool und wird derzeit nur vom SyringeExtruder (Child) aufgerufen
IF pTool^.P_eObjectType = E_ObjectType.OBJECTTYPE_Extruder THEN
	nSlotDiff :=  UINT_TO_INT(pToolSlot^.P_nNr) - UINT_TO_INT(nMasterSlotNr);
	nAxisNr := pZAxisRef^.nChannel + nSlotDiff * 2; //Es muss immer eine freie Achse dazwischen sein.
	M_GetZAxisRef := ADR(pFbMultiZ^.aFbZAxisRef[nAxisNr]);
	IF M_GetZAxisRef^.eDetectedToolType <> E_MzToolType.TOOL_TYPE_SyringeExtruder THEN
		M_GetZAxisRef := 0;
	END_IF
ELSE
	M_GetZAxisRef := SUPER^.M_GetZAxisRef(pTool, pParentSlot);
END_IF
END_METHOD

METHOD M_Prepare : ST_MethResult
VAR_INPUT
	bExecute : BOOL;
END_VAR

VAR
 	i : USINT;	
END_VAR

VAR_INST
	nState : USINT;	
END_VAR
IF bExecute THEN
	IF nState = 0 THEN
		nState := 80;
		FOR i := 1 TO 3 BY 1 DO
			IF aiDispenser[i] <> 0 THEN
				M_Prepare.nErrorId := aiDispenser[i].M_DispenserPrepare();
				IF M_Prepare.nErrorId > 0 THEN
					M_Prepare.bError := TRUE;
					M_Prepare.bBusy := FALSE;
					RETURN;
				END_IF
				IF aiDispenser[i].P_eDispenserState = E_DispenserState.Preparing THEN
					nState := 1;
					M_Prepare.bBusy := TRUE;				
					RETURN;
				END_IF
			END_IF
		END_FOR
	ELSIF nState = 1 THEN
		FOR i := 1 TO 3 BY 1 DO
			IF aiDispenser[i] <> 0 THEN
				IF aiDispenser[i].P_bError THEN
					M_Prepare.bError := TRUE;
					M_Prepare.bBusy := FALSE;
					RETURN;
				END_IF
				IF aiDispenser[i].P_eDispenserState = E_DispenserState.Preparing THEN
					nState := 1;
					M_Prepare.bBusy := TRUE;
					RETURN;
				END_IF				
			END_IF
		END_FOR
	END_IF
ELSE
	nState := 0;	
END_IF
END_METHOD

METHOD M_SetAllProps : ERRORID
VAR_INPUT
	refCmdData : REFERENCE TO  ST_CmdData;
END_VAR
M_SetAllProps := SUPER^.M_SetAllProps(refCmdData);

IF M_SetAllProps > 0 THEN
	RETURN;
END_IF

nCurrentPropIndex := nCurrentPropIndex + 1;
nSpecPropIndex := nCurrentPropIndex;
nMasterSlotNr := DINT_TO_USINT(refCmdData.n32Data[nCurrentPropIndex]);
nNoOfProps := nCurrentPropIndex + 1;
END_METHOD

METHOD M_SetPrintParams : ST_MethResult
VAR_INPUT
	eType 		: E_PrintParamType;
	nNumerator	: USINT;
	nValue		: DINT;
END_VAR

